Yaskawa INFORM job: X2_29-32(-90,180)_HARDOX.JBI

/JOB
//NAME X2_29-32(-90,180)_HARDOX
//POS
///NPOS 464,464,464,30,0,0
///TOOL 0
///POSTYPE PULSE
///PULSE
C00000=2000,-95440,-72516,0,38121,0
C00001=-80443,-95440,-72516,-46202,38121,50067
C00002=-52411,-63190,-65629,-41206,65263,51508
C00003=-73087,-23788,-54178,-20049,70640,39353
C00004=-137855,-58890,-63164,50426,57117,3007
C00005=-121629,-1819,-23267,32035,72941,16834
C00006=-120935,3126,-16373,32060,71231,16611
C00007=-120668,5150,-13541,32087,70531,16512
C00008=-120826,7275,-11699,32150,70554,16454
C00009=-120668,5150,-13541,32087,70531,16512
C00010=-120649,6560,-12069,32112,70369,16472
C00011=-120645,6560,-10825,32251,69714,16277
C00012=-120649,6560,-12069,32112,70369,16472
C00013=-120913,4529,-14922,32082,71075,16573
C00014=-121602,-429,-21862,32048,72802,16805
C00015=-120074,-1541,-23154,10906,71264,22392
C00016=-120462,3262,-16191,11181,69532,22093
C00017=-120612,5232,-13331,11295,68818,21971
C00018=-120770,7357,-11488,11363,68799,21912
C00019=-120612,5232,-13331,11295,68818,21971
C00020=-120702,6360,-12382,11332,68826,21940
C00021=-120699,6356,-11141,11388,68075,21868
C00022=-120702,6360,-12382,11332,68826,21940
C00023=-120555,4389,-15254,11219,69547,22062
C00024=-120172,-412,-22245,10944,71297,22361
C00025=-149351,-10161,-47708,21219,87013,14604
C00026=-137351,69022,23166,10145,93880,-87530
C00027=-140356,69806,28572,10729,91371,-88714
C00028=-140356,69507,29335,10724,90759,-88767
C00029=-140356,69553,29212,10724,90856,-88758
C00030=-140261,66601,25742,10710,91452,-88676
C00031=-140356,69553,29212,10724,90856,-88758
C00032=-136478,56234,14982,2602,86089,-89060
C00033=-137167,55940,14650,2804,86164,-89279
C00034=-140356,69877,28402,10731,91510,-88702
C00035=-138692,40861,2416,14344,76332,-89060
C00036=-138692,40492,3371,14387,75578,-89150
C00037=-138692,40531,3265,14382,75660,-89140
C00038=-138845,42877,5737,14463,75381,-89226
C00039=-138692,40531,3265,14382,75660,-89140
C00040=-137711,40836,3584,13981,75458,-88832
C00041=-137936,41046,2771,14040,76086,-88835
C00042=-125437,22929,-16002,8654,76643,-84658
C00043=-125437,22691,-15519,8668,76228,-84687
C00044=-125436,22336,-14745,8692,75581,-84731
C00045=-125436,22385,-14855,8689,75673,-84725
C00046=-125647,22419,-14823,8780,75693,-84793
C00047=-125456,22816,-15761,8671,76446,-84677
C00048=-124626,66836,21249,8312,76213,-84427
C00049=-124626,66325,22111,8339,75427,-84480
C00050=-124626,66371,22030,8336,75501,-84476
C00051=-124784,66398,22063,8405,75510,-84527
C00052=-124718,66903,21186,8350,76294,-84452
C00053=-140356,71956,24660,10787,94825,-88416
C00054=-145256,112136,75534,11701,85011,-90920
C00055=-134601,86997,59569,9608,80583,-87665
C00056=-133445,96084,71731,8965,80046,-87331
C00057=-133445,96731,74588,9003,78636,-87434
C00058=-133445,96669,74335,9000,78758,-87425
C00059=-133228,92094,68499,8930,79959,-87263
C00060=-133445,96669,74335,9000,78758,-87425
C00061=-133796,95310,72593,9053,79166,-87516
C00062=-134289,94368,71392,9135,79474,-87664
C00063=-133445,96257,72553,8977,79632,-87361
C00064=-124701,59773,45425,12728,59446,-85623
C00065=-124701,60369,47958,12892,58224,-85768
C00066=-124701,60307,47711,12875,58342,-85755
C00067=-125124,62964,50756,13140,57912,-85979
C00068=-124701,60307,47711,12875,58342,-85755
C00069=-124156,61205,48739,12645,58092,-85564
C00070=-123633,62204,49884,12428,57822,-85386
C00071=-124701,59815,45622,12740,59350,-85635
C00072=-140824,71424,26731,-14708,78728,-67313
C00073=-138566,88921,46332,-15736,76162,-66229
C00074=-147570,88381,37329,-2994,91316,-68707
C00075=-150504,94687,46185,-534,91721,-69351
C00076=-150504,94129,46947,-534,90966,-69348
C00077=-150505,94206,46833,-534,91077,-69347
C00078=-150278,92960,45244,-584,91415,-69274
C00079=-150242,94003,44864,-592,92185,-69267
C00080=-154498,83968,32184,366,94826,-70609
C00081=-154498,83134,33047,365,93865,-70611
C00082=-154498,83201,32975,365,93945,-70611
C00083=-154422,82409,31994,348,94142,-70584
C00084=-154454,83590,32320,355,94549,-70593
C00085=-163409,96576,47553,1962,92625,-73499
C00086=-157730,108398,64416,-12689,90385,-74066
C00087=-157730,108035,65300,-12685,89672,-73993
C00088=-157730,108081,65179,-12685,89767,-74003
C00089=-157935,107012,63772,-12649,90048,-74099
C00090=-157741,107169,62938,-12691,90658,-74096
C00091=-153583,44731,-17162,-14334,108038,-74686
C00092=-119941,-49108,-60020,12756,52739,20459
C00093=-119789,-74783,-79746,11606,60570,21449
C00094=-121427,-115493,-86071,-971,23186,13
C00095=-103613,-33005,-61039,-35202,65094,-22685
C00096=-106311,42726,-13762,-25892,102641,-65108
C00097=-107595,62330,8123,-25246,99218,-64778
C00098=-113201,64656,7277,-4573,99753,-62165
C00099=-113587,63448,8349,-4464,98459,-62235
C00100=-113587,62765,8896,-4459,97772,-62209
C00101=-113587,62841,8834,-4460,97849,-62212
C00102=-113249,60648,6293,-4545,98301,-62127
C00103=-113587,62841,8834,-4460,97849,-62212
C00104=-104619,65495,14505,-22863,97888,-62863
C00105=-105135,64543,13388,-22764,97939,-63047
C00106=-113587,63726,8142,-4473,98728,-62244
C00107=-108677,35532,-14553,-8240,80429,-60363
C00108=-108677,34745,-13725,-8259,79524,-60302
C00109=-108677,34861,-13853,-8256,79661,-60312
C00110=-109185,36959,-11698,-8032,79365,-60451
C00111=-108678,34861,-13851,-8256,79664,-60311
C00112=-108199,35754,-12936,-8475,79600,-60161
C00113=-107535,36718,-11943,-8775,79549,-59951
C00114=-108678,35482,-14504,-8241,80378,-60358
C00115=-107675,14693,-34978,-8652,82358,-60193
C00116=-103613,-33005,-61039,-35202,65094,-22685
C00117=-118652,-1130,-18887,-50959,75871,-22344
C00118=-120065,3095,-12579,-50928,73991,-22034
C00119=-120612,5858,-10323,-50783,73711,-22168
C00120=-120794,7716,-8707,-50742,73586,-22192
C00121=-120612,6719,-9575,-50786,73699,-22162
C00122=-120612,6754,-8612,-50907,73330,-21953
C00123=-120612,6719,-9575,-50786,73699,-22162
C00124=-120164,4326,-11494,-50910,73914,-22043
C00125=-118762,92,-17836,-50934,75798,-22362
C00126=-120082,-2017,-23568,-21020,76850,-12939
C00127=-120471,2786,-16617,-21041,75059,-12760
C00128=-120621,6055,-13261,-21027,74660,-12744
C00129=-120866,7545,-11965,-20950,74569,-12818
C00130=-120698,6523,-12855,-21003,74632,-12768
C00131=-120698,6506,-12245,-21039,74273,-12705
C00132=-120698,6523,-12855,-21003,74632,-12768
C00133=-120547,3972,-15593,-21018,75020,-12781
C00134=-120163,-831,-22574,-20994,76828,-12964
C00135=-120068,-2141,-23641,-4094,79360,4817
C00136=-120458,2664,-16692,-4000,77538,4745
C00137=-120609,5664,-13523,-3960,77123,4708
C00138=-120915,7025,-12341,-3868,77081,4605
C00139=-120609,5664,-13523,-3960,77123,4708
C00140=-120609,5646,-12752,-3962,76640,4725
C00141=-120609,5664,-13523,-3960,77123,4708
C00142=-120559,4206,-15421,-3970,77544,4711
C00143=-120175,-595,-22406,-4061,79389,4780
C00144=-120687,14813,-21149,-8531,87328,5298
C00145=-120686,13947,-18988,-8540,85572,5418
C00146=-121162,15330,-17687,-8405,85435,5272
C00147=-120827,14308,-18485,-8500,85444,5381
C00148=-120926,18777,-11948,-23218,84672,-11491
C00149=-120686,12805,-15419,-25390,80631,-12632
C00150=-120686,13423,-17789,-25296,82244,-12980
C00151=-103613,-33005,-61039,-35202,65094,-22685
C00152=-106311,42726,-13762,-25892,102641,-65108
C00153=-107595,62330,8123,-25246,99218,-64778
C00154=-113201,64656,7277,-4573,99753,-62165
C00155=-140379,75416,22801,13293,101526,-67991
C00156=-140410,74339,22937,13264,100908,-68069
C00157=-136164,75986,24927,12542,99919,-66800
C00158=-136164,75986,24927,12542,99919,-66800
C00159=-130307,51965,-280,1869,88480,-68213
C00160=-130096,37123,-11525,-190,78489,-68727
C00161=-129173,33980,-14136,-6116,77606,-69795
C00162=-117721,30667,-17043,-13656,78654,-66867
C00163=-117721,30667,-17043,-13656,78654,-66867
C00164=-116349,51111,-1470,-15144,92480,-68252
C00165=-140410,74339,22937,13264,100908,-68069
C00166=-140394,75226,22544,13300,101585,-67989
C00167=-143024,47479,-9541,14128,107315,-68172
C00168=-103613,-33005,-61039,-35202,65094,-22685
C00169=-121427,-115493,-86071,-971,23186,13
C00170=-119789,-74783,-79746,11606,60570,21449
C00171=-119941,-49108,-60020,12756,52739,20459
C00172=-140276,36725,370,11673,88260,-76470
C00173=-134601,86997,59569,9608,80583,-87665
C00174=-138207,103684,77785,17301,84049,-88284
C00175=-137334,101091,76947,17225,83081,-88111
C00176=-133753,108880,87117,16824,80164,-87228
C00177=-133753,108880,87117,16824,80164,-87228
C00178=-134207,73969,56380,20261,66539,-89438
C00179=-133045,60996,43275,16271,60703,-90304
C00180=-131571,55694,36295,8271,61065,-90068
C00181=-118397,49989,30000,-2055,61299,-85309
C00182=-118397,49989,30000,-2055,61299,-85309
C00183=-130531,95421,68229,8568,83299,-86105
C00184=-137334,101091,76947,17225,83081,-88111
C00185=-137309,103311,78077,17211,83503,-88042
C00186=-146018,96073,47329,18619,99857,-88679
C00187=-146906,94555,49940,18578,97784,-89305
C00188=-142933,95333,50973,18069,96712,-88106
C00189=-142933,95333,50973,18069,96712,-88106
C00190=-142636,61819,14681,18419,84430,-90138
C00191=-141138,57519,10350,14135,81366,-90943
C00192=-124192,48626,472,-4337,80868,-88195
C00193=-120975,45190,-1140,-14592,79533,-89080
C00194=-120975,45190,-1140,-14592,79533,-89080
C00195=-121205,42490,-4021,-14479,79869,-89194
C00196=-146906,94555,49940,18578,97784,-89305
C00197=-146868,95992,48950,18656,99055,-89096
C00198=-148689,99526,52175,12058,97492,78019
C00199=-152884,101141,55717,10807,87410,75244
C00200=-156822,87647,42567,16335,79952,73793
C00201=-156347,101107,61134,16633,80023,73987
C00202=-156384,100515,60368,16637,80191,73997
C00203=-156384,100515,60368,16637,80191,73997
C00204=-156439,104263,64294,16482,82615,74284
C00205=-153753,110748,70719,9837,85116,74669
C00206=-150674,104620,59635,-3355,94991,76839
C00207=-155137,96651,49130,-4365,100310,75004
C00208=-155137,96651,49130,-4365,100310,75004
C00209=-157583,94336,46084,-1766,101365,64930
C00210=-158276,84861,34738,-3244,98222,56321
C00211=-159116,67672,17693,-4464,87885,55617
C00212=-158508,68290,14812,-4659,90001,55728
C00213=-159737,63424,5379,-4280,93236,55245
C00214=-162760,44138,-13287,27476,96226,62089
C00215=-135421,18423,-39272,17962,92414,69811
C00216=-134350,548,-53000,17534,91515,69996
C00217=-134346,591,-47047,17501,88033,69498
C00218=-133581,11899,-36465,17450,85821,69480
C00219=-133633,12580,-37298,17464,86638,69580
C00220=-133478,14153,-35291,17454,85907,69536
C00221=-130266,45661,-10200,12167,104064,71599
C00222=-133264,15600,-32829,17378,85127,69491
C00223=-130716,70167,29007,18289,68146,68029
C00224=-130765,70515,28279,18240,68753,68107
C00225=-130672,73101,31358,18260,68194,68051
C00226=-130688,71478,30626,18340,67728,67974
C00227=-130258,88127,52093,19258,61489,67116
C00228=-130258,88603,49705,18973,63112,67401
C00229=-136006,-18137,-67664,18160,91268,69467
C00230=-130548,-59686,-65936,20231,53139,15983
C00231=-120686,14413,-19191,15888,76861,21657
C00232=-120686,13677,-16924,15998,75153,21431
C00233=-120864,13854,-15557,16118,74464,21280
C00234=-120686,13319,-15964,16052,74414,21331
C00235=-120685,12972,2532,58159,63782,21773
C00236=-120685,12849,1627,57961,64053,21984
C00237=-120685,12557,-1021,57383,64873,22611
C00238=-118042,2496,-28680,21493,77866,23942
C00239=-119941,-49108,-60020,12756,52739,20459
C00240=-119789,-74783,-79746,11606,60570,21449
C00241=-121427,-115493,-86071,-971,23186,13
C00242=-103613,-33005,-61039,-35202,65094,-22685
C00243=-134099,37898,13128,-30528,62935,-29291
C00244=-134100,37844,14655,-30775,62096,-29040
C00245=-131820,39720,18358,-33617,61933,-27865
C00246=-133865,38946,16955,-31235,61462,-28734
C00247=-133724,38989,23896,-55752,81870,-5528
C00248=-134106,38309,22847,-57056,83615,-3951
C00249=-130543,37429,19989,-57378,86491,-3781
C00250=-124532,-28339,-37080,2656,37858,63256
C00251=-80443,-95440,-72516,-46202,38121,50067
C00252=-628,-74499,-67639,-57475,89722,72456
C00253=3643,-76224,-106676,19950,71810,76872
C00254=-57022,-39792,-97587,-14580,73098,62715
C00255=-77894,6609,-39652,-10081,68656,55583
C00256=-79326,8848,-34628,-9340,66588,55287
C00257=-79882,9812,-32559,-9051,65763,55166
C00258=-80655,11957,-30643,-8578,65611,54918
C00259=-79882,9812,-32559,-9051,65763,55166
C00260=-80541,11612,-30977,-8647,65649,54954
C00261=-80539,10894,-29907,-8717,64633,55031
C00262=-80541,11612,-30977,-8647,65649,54954
C00263=-79996,10638,-33064,-8931,66478,55073
C00264=-78593,8374,-38132,-9661,68553,55366
C00265=-77879,6415,-39661,-10096,68566,55596
C00266=-79312,8664,-34633,-9354,66499,55298
C00267=-79868,9631,-32562,-9065,65674,55178
C00268=-80642,11778,-30647,-8592,65523,54929
C00269=-79868,9631,-32562,-9065,65674,55178
C00270=-80486,11377,-31039,-8686,65573,54978
C00271=-80483,10662,-29965,-8757,64557,55056
C00272=-80486,11377,-31039,-8686,65573,54978
C00273=-79940,10400,-33127,-8971,66401,55097
C00274=-78534,8129,-38197,-9702,68474,55392
C00275=-80101,2636,-42462,-8765,68121,54914
C00276=-81514,5018,-37368,-8012,66098,54596
C00277=-82062,6036,-35274,-7718,65291,54467
C00278=-82824,8247,-33345,-7247,65177,54218
C00279=-82062,6036,-35274,-7718,65291,54467
C00280=-82687,7884,-33751,-7328,65251,54260
C00281=-82684,7173,-32662,-7390,64223,54326
C00282=-82687,7884,-33751,-7328,65251,54260
C00283=-82150,6860,-35861,-7618,66062,54387
C00284=-80765,4464,-40992,-8359,68092,54701
C00285=-102565,-17528,-58279,5105,67037,47705
C00286=-103540,-14129,-52689,5779,65410,47308
C00287=-103914,-12731,-50412,6044,64755,47149
C00288=-104433,-9984,-48291,6364,64897,46981
C00289=-103914,-12731,-50412,6044,64755,47149
C00290=-104359,-10402,-48741,6314,64954,47009
C00291=-104354,-11138,-47602,6366,63880,46952
C00292=-104359,-10402,-48741,6314,64954,47009
C00293=-103995,-11787,-51026,6054,65619,47167
C00294=-103047,-15149,-56634,5395,67274,47560
C00295=-80233,11979,-33534,-13378,69985,55632
C00296=-80229,10556,-31784,-13533,68226,55836
C00297=-80227,10062,-31089,-13596,67561,55913
C00298=-85904,3072,-37201,-10254,66968,54061
C00299=-91604,-2565,-41777,-6847,66341,52198
C00300=-101176,-9655,-47350,-1032,65699,49019
C00301=-100886,-9155,-48096,-1203,66417,49108
C00302=-100216,-7271,-49632,-1590,68341,49304
C00303=-80300,11336,-32181,-3939,63811,54132
C00304=-80297,10024,-30348,-4003,62013,54196
C00305=-80296,9579,-29637,-4028,61349,54220
C00306=-80356,9883,-29495,-3999,61418,54197
C00307=-80338,10281,-30338,-3972,62137,54177
C00308=-80341,11605,-32161,-3909,63935,54114
C00309=-57022,-39792,-97587,-14580,73098,62715
C00310=-628,-74499,-67639,-57475,89722,72456
C00311=-628,-74499,-67639,-57475,89722,72456
C00312=-616,-75233,-71189,-57531,90735,71761
C00313=3643,-76224,-106674,19950,71813,76873
C00314=-42730,11015,-70691,-38334,96086,2936
C00315=-63606,9545,-60534,-45336,92087,-16638
C00316=-78956,5069,-41799,-36523,82652,-30708
C00317=-79715,8164,-36018,-36343,80767,-30358
C00318=-80007,9457,-33651,-36288,80012,-30216
C00319=-80417,12097,-31285,-36126,79775,-30292
C00320=-80007,9457,-33651,-36288,80012,-30216
C00321=-80344,11698,-31669,-36153,79828,-30282
C00322=-80337,10939,-30633,-36254,78993,-30001
C00323=-80344,11698,-31669,-36153,79828,-30282
C00324=-80059,10405,-34052,-36203,80590,-30428
C00325=-79319,7312,-39869,-36371,82488,-30786
C00326=-78994,5332,-41692,-36502,82694,-30736
C00327=-79751,8420,-35912,-36322,80808,-30385
C00328=-80043,9710,-33546,-36267,80051,-30242
C00329=-80452,12349,-31177,-36105,79813,-30317
C00330=-80043,9710,-33546,-36267,80051,-30242
C00331=-80378,11838,-31671,-36133,79874,-30310
C00332=-80371,11075,-30637,-36233,79039,-30029
C00333=-80378,11838,-31671,-36133,79874,-30310
C00334=-80093,10547,-34052,-36183,80637,-30456
C00335=-79355,7462,-39866,-36352,82536,-30815
C00336=-79090,5824,-41546,-36452,82791,-30803
C00337=-79842,8894,-35770,-36272,80900,-30451
C00338=-80133,10177,-33405,-36216,80142,-30307
C00339=-80539,12815,-31031,-36055,79902,-30380
C00340=-80133,10177,-33405,-36216,80142,-30307
C00341=-80467,12378,-31515,-36079,79989,-30382
C00342=-80461,11606,-30490,-36178,79153,-30101
C00343=-80467,12378,-31515,-36079,79989,-30382
C00344=-80184,11095,-33894,-36130,80753,-30529
C00345=-79450,8031,-39703,-36300,82657,-30890
C00346=-79130,5997,-41490,-36432,82820,-30827
C00347=-79881,9061,-35715,-36251,80928,-30474
C00348=-80171,10342,-33350,-36196,80169,-30330
C00349=-80577,12980,-30974,-36035,79928,-30403
C00350=-80171,10342,-33350,-36196,80169,-30330
C00351=-80499,12601,-31443,-36059,80034,-30409
C00352=-80493,11826,-30422,-36158,79199,-30129
C00353=-80499,12601,-31443,-36059,80034,-30409
C00354=-80216,11321,-33822,-36110,80799,-30556
C00355=-79484,8265,-39628,-36281,82705,-30918
C00356=-80360,13355,-34008,-31162,79863,-31191
C00357=-80358,11846,-32319,-31320,78301,-30757
C00358=-80129,11573,-31352,-31494,77744,-30518
C00359=-80458,11751,-31298,-31342,77685,-30622
C00360=-80398,12063,-32232,-31297,78337,-30782
C00361=-80400,13577,-33916,-31139,79899,-31215
C00362=-80289,11819,-32883,-40833,82428,-30239
C00363=-80286,10439,-31086,-40975,81039,-29694
C00364=-80284,9940,-30341,-41041,80492,-29477
C00365=-80262,9799,-30343,-41055,80447,-29451
C00366=-80245,10226,-31168,-40996,81011,-29666
C00367=-80248,11601,-32971,-40853,82401,-30212
C00368=-66712,19655,-58640,-43457,90055,-24381
C00369=-33423,17994,-60377,-60627,102988,-19600
C00370=-628,-74499,-67639,-57475,89722,-77289
C00371=-111516,-94989,-87682,-11539,41033,-8318
C00372=-107125,-12532,-46236,-32676,64375,-10703
C00373=-119952,37605,6162,-31233,75137,-17424
C00374=-120511,42562,14108,-31354,72919,-17016
C00375=-120728,44654,17433,-31427,72005,-16841
C00376=-120598,46946,19889,-31526,71766,-16719
C00377=-120728,44654,17433,-31427,72005,-16841
C00378=-120690,45788,18679,-31469,71861,-16784
C00379=-120687,45721,19851,-31594,71213,-16595
C00380=-120690,45788,18679,-31469,71861,-16784
C00381=-120474,43679,15324,-31394,72783,-16962
C00382=-119917,38688,7316,-31265,75018,-17376
C00383=-121235,29127,929,-10497,72605,-22385
C00384=-120892,33963,8709,-10768,70384,-22067
C00385=-120760,35995,11952,-10883,69467,-21936
C00386=-120625,38237,14258,-10956,69222,-21864
C00387=-120760,35995,11952,-10883,69467,-21936
C00388=-120657,37146,13206,-10937,69303,-21884
C00389=-120654,37124,14427,-10991,68554,-21813
C00390=-120657,37146,13206,-10937,69303,-21884
C00391=-120788,35099,9935,-10821,70230,-22016
C00392=-121127,30229,2096,-10548,72470,-22335
C00393=-114017,-48711,-62992,-16459,47417,-13874
C00394=-111516,-94989,-87682,-11539,41033,-8318
C00395=-126605,-77887,-93073,32833,63422,15189
C00396=-122507,12852,-43627,17515,100315,22769
C00397=-122731,-562,-19309,51196,76332,22742
C00398=-121309,3590,-13049,51151,74446,22427
C00399=-120759,5312,-10468,51156,73690,22291
C00400=-120602,7442,-8613,51127,73573,22309
C00401=-120759,5312,-10468,51156,73690,22291
C00402=-120666,6547,-9361,51143,73609,22295
C00403=-120662,6597,-8073,51308,73115,22013
C00404=-120666,6547,-9361,51143,73609,22295
C00405=-121212,4820,-11958,51134,74367,22434
C00406=-122622,659,-18251,51172,76257,22758
C00407=-122507,10859,-42333,17402,98575,22516
C00408=-121302,-1391,-23074,21379,77148,13095
C00409=-120901,3377,-16122,21398,75339,12912
C00410=-120747,5333,-13267,21416,74597,12833
C00411=-120590,7459,-11416,21370,74514,12875
C00412=-120747,5333,-13267,21416,74597,12833
C00413=-120673,6521,-12221,21396,74547,12851
C00414=-120670,6504,-10992,21468,73832,12721
C00415=-120673,6521,-12221,21396,74547,12851
C00416=-120826,4563,-15090,21376,75296,12931
C00417=-121222,-206,-22073,21354,77121,13119
C00418=-121314,-1652,-23262,4485,79740,-4708
C00419=-120913,3117,-16316,4391,77900,-4639
C00420=-120758,5074,-13462,4356,77144,-4613
C00421=-120601,7199,-11615,4311,77090,-4561
C00422=-120758,5074,-13462,4356,77144,-4613
C00423=-120661,6618,-12165,4328,77134,-4580
C00424=-120658,6600,-10936,4339,76370,-4606
C00425=-120661,6618,-12165,4328,77134,-4580
C00426=-120814,4660,-15035,4362,77900,-4605
C00427=-121209,-107,-22019,4454,79763,-4672
C00428=-120687,46979,12625,8958,83453,-5452
C00429=-120687,46939,12852,8960,83294,-5464
C00430=-121610,47377,14332,9229,82719,-5809
C00431=-120687,46779,13614,8967,82756,-5503
C00432=-120687,46744,18453,25999,77793,12121
C00433=-120687,46348,16793,25935,78533,12285
C00434=-120687,46750,14296,25811,80109,12635
C00435=-133650,-5326,-40947,35821,67459,4738
C00436=-126605,-79487,-84548,34660,58331,13454
C00437=-111516,-94989,-87682,-11539,41033,-8318
C00438=-114017,-48711,-62992,-16459,47417,-13874
C00439=-117875,8541,-26754,-15356,68464,-18868
C00440=-120687,46680,12303,-15684,74586,-21239
C00441=-120687,46183,14573,-15804,72993,-21028
C00442=-120687,45847,15503,-15862,72274,-20933
C00443=-120687,45820,15711,-15860,72146,-20914
C00444=-120686,46430,31549,-51889,62431,-21622
C00445=-120686,46225,30262,-51616,62867,-21897
C00446=-120686,45862,27317,-50999,63909,-22538
C00447=-117875,8541,-26754,-15356,68464,-18868
C00448=-114017,-48711,-62992,-16459,47417,-13874
C00449=-111516,-94989,-87682,-11539,41033,-8318
C00450=-126605,-79487,-84548,34660,58331,13454
C00451=-133650,-5326,-40947,35821,67459,4738
C00452=-107292,16964,-8341,30286,65218,30077
C00453=-107291,16711,-5651,30703,63668,29626
C00454=-107319,17056,-4163,30899,63039,29427
C00455=-107325,17150,-4064,30903,63037,29424
C00456=-107531,17120,3962,56911,83437,5110
C00457=-107292,16975,3345,57479,84239,4502
C00458=-107292,16775,1094,57407,84952,4997
C00459=-118083,23631,-28824,25815,115568,5891
C00460=-116334,-45445,-82386,24519,90130,1359
C00461=-114916,-111439,-107393,23774,54945,-5331
C00462=-628,-74499,-67639,-57475,89722,-77289
C00463=2000,17994,-60377,0,102988,0
BC00000=30861,666204,744559
BC00001=125925,693938,117612
BC00002=171995,715848,96803
BC00003=199966,729151,84169
BC00004=289373,771673,43785
BC00005=289373,771673,43785
BC00006=289373,771673,43785
BC00007=289373,771673,43785
BC00008=289373,771673,43785
BC00009=289373,771673,43785
BC00010=289373,771673,43785
BC00011=289373,771673,43785
BC00012=289373,771673,43785
BC00013=289373,771673,43785
BC00014=289373,771673,43785
BC00015=275430,758658,78312
BC00016=275430,758658,78312
BC00017=275430,758658,78312
BC00018=275430,758658,78312
BC00019=275430,758658,78312
BC00020=275430,758658,78312
BC00021=275430,758658,78312
BC00022=275430,758658,78312
BC00023=275430,758658,78312
BC00024=275430,758658,78312
BC00025=343308,785974,78310
BC00026=343308,785974,78310
BC00027=343308,785974,78310
BC00028=343308,785974,78310
BC00029=343308,785974,78310
BC00030=343308,785974,78310
BC00031=343308,785974,78310
BC00032=343308,785974,78310
BC00033=343308,785974,78310
BC00034=343308,785974,78310
BC00035=343308,785974,78310
BC00036=343308,785974,78310
BC00037=343308,785974,78310
BC00038=343308,785974,78310
BC00039=343308,785974,78310
BC00040=343308,785974,78310
BC00041=343308,785974,78310
BC00042=318074,785974,78310
BC00043=318074,785974,78310
BC00044=318074,785974,78309
BC00045=318074,785974,78309
BC00046=318074,785974,78309
BC00047=318074,785974,78309
BC00048=318074,785624,15543
BC00049=318074,785624,15543
BC00050=318074,785624,15543
BC00051=318074,785624,15543
BC00052=318074,785624,15543
BC00053=343308,785974,78310
BC00054=370182,760337,78310
BC00055=370182,760337,184963
BC00056=370182,760337,157808
BC00057=370182,760337,157808
BC00058=370182,760337,157808
BC00059=370182,760337,157808
BC00060=370182,760337,157808
BC00061=370182,760337,157808
BC00062=370182,760337,157808
BC00063=370182,760337,157808
BC00064=340749,760337,227440
BC00065=340749,760337,227440
BC00066=340749,760337,227440
BC00067=340749,760337,227440
BC00068=340749,760337,227440
BC00069=340749,760337,227440
BC00070=340749,760337,227440
BC00071=340749,760337,227440
BC00072=340750,760338,77389
BC00073=340750,760338,30516
BC00074=348215,785472,13
BC00075=348215,785472,13
BC00076=348215,785471,10
BC00077=348215,785471,9
BC00078=348215,785471,9
BC00079=348215,785471,9
BC00080=348215,785471,9
BC00081=348215,785471,9
BC00082=348215,785471,9
BC00083=348215,785471,9
BC00084=348215,785471,9
BC00085=370537,785471,9
BC00086=370537,785471,9
BC00087=370537,785471,9
BC00088=370537,785471,9
BC00089=370537,785471,9
BC00090=370537,785471,9
BC00091=370537,785471,9
BC00092=275430,725446,78312
BC00093=275430,674753,78312
BC00094=160005,679271,117612
BC00095=134493,734471,53
BC00096=134493,734471,4
BC00097=134493,734471,4
BC00098=134493,734471,4
BC00099=134493,734471,4
BC00100=134493,734471,4
BC00101=134493,734471,4
BC00102=134493,734471,4
BC00103=134493,734471,4
BC00104=134493,734471,4
BC00105=134493,734471,4
BC00106=134493,734471,4
BC00107=134493,734471,4
BC00108=134493,734471,4
BC00109=134493,734471,4
BC00110=134493,734471,4
BC00111=134494,734471,1
BC00112=134493,734471,4
BC00113=134493,734471,4
BC00114=134494,734471,1
BC00115=134493,734471,4
BC00116=134493,734471,53
BC00117=134493,734471,53
BC00118=134493,734471,53
BC00119=134493,734471,53
BC00120=134493,734471,53
BC00121=134493,734471,53
BC00122=134493,734471,53
BC00123=134493,734471,53
BC00124=134493,734471,53
BC00125=134493,734471,53
BC00126=120013,731989,63282
BC00127=120013,731989,63282
BC00128=120013,731989,63282
BC00129=120013,731989,63282
BC00130=120013,731989,63282
BC00131=120013,731989,63282
BC00132=120013,731989,63282
BC00133=120013,731989,63282
BC00134=120013,731989,63282
BC00135=143296,743099,87341
BC00136=143296,743099,87341
BC00137=143296,743099,87341
BC00138=143296,743099,87341
BC00139=143296,743099,87341
BC00140=143296,743099,87341
BC00141=143296,743099,87341
BC00142=143296,743099,87341
BC00143=143296,743099,87341
BC00144=160875,733218,0
BC00145=159215,738452,0
BC00146=159050,738970,0
BC00147=154263,739676,0
BC00148=124438,729775,0
BC00149=121804,726587,0
BC00150=123464,721353,0
BC00151=134493,734471,53
BC00152=134493,734471,4
BC00153=134493,734471,4
BC00154=134493,734471,4
BC00155=202496,734468,2
BC00156=202496,734468,2
BC00157=202496,734468,2
BC00158=202496,734468,2
BC00159=202496,734468,2
BC00160=202496,734468,2
BC00161=202496,734468,2
BC00162=167019,734468,2
BC00163=167019,734468,2
BC00164=163805,734468,2
BC00165=202496,734468,2
BC00166=202496,734468,2
BC00167=202496,734468,2
BC00168=134493,734471,53
BC00169=160005,679271,117612
BC00170=275430,674753,78312
BC00171=275430,725446,78312
BC00172=359023,756228,172403
BC00173=370182,760337,184963
BC00174=370182,760337,129528
BC00175=370181,760337,129525
BC00176=370055,760318,129428
BC00177=370055,760318,129428
BC00178=370055,760499,186673
BC00179=370055,760499,186673
BC00180=369975,760487,186584
BC00181=327884,760487,186584
BC00182=327884,760487,186584
BC00183=355542,760337,129525
BC00184=370181,760337,129525
BC00185=370181,760337,129525
BC00186=355947,779528,6445
BC00187=356286,779072,9376
BC00188=356321,779025,9678
BC00189=356321,779025,9678
BC00190=356321,779025,9678
BC00191=356321,779025,9727
BC00192=316277,778464,10141
BC00193=316277,778464,10141
BC00194=316277,778464,10141
BC00195=316277,778464,10141
BC00196=356286,779072,9376
BC00197=356286,779072,9376
BC00198=356286,779072,9376
BC00199=356286,779072,9376
BC00200=356286,779072,9376
BC00201=356286,779072,9376
BC00202=356286,779072,9376
BC00203=356286,779072,9376
BC00204=356286,779072,9376
BC00205=356286,779072,9376
BC00206=359300,795873,31
BC00207=359300,795873,31
BC00208=359300,795873,31
BC00209=359300,795873,31
BC00210=359300,795873,31
BC00211=359300,795873,31
BC00212=359300,795873,31
BC00213=359300,795873,31
BC00214=359300,795873,31
BC00215=329302,795872,29
BC00216=329302,795872,29
BC00217=329302,795872,29
BC00218=329622,793366,28
BC00219=329626,793338,28
BC00220=329692,792815,28
BC00221=329692,792815,28
BC00222=329692,792815,28
BC00223=331278,780389,22
BC00224=331278,780389,22
BC00225=331278,780389,22
BC00226=331302,780203,22
BC00227=331702,777069,20
BC00228=331702,777069,20
BC00229=329302,795872,29
BC00230=311672,797875,78800
BC00231=261630,745054,0
BC00232=261335,750526,0
BC00233=262635,752963,0
BC00234=310200,761264,0
BC00235=269037,768534,0
BC00236=267560,766459,0
BC00237=263869,761272,0
BC00238=263869,761272,0
BC00239=275430,725446,78312
BC00240=275430,674753,78312
BC00241=160005,679271,117612
BC00242=134493,734471,53
BC00243=177141,688062,0
BC00244=175480,693296,0
BC00245=174817,695179,178
BC00246=160472,692881,15
BC00247=152915,732429,1
BC00248=154775,734615,0
BC00249=161011,731782,0
BC00250=160005,693938,117612
BC00251=125925,693938,117612
BC00252=97174,666880,426359
BC00253=199464,674570,1075173
BC00254=48447,721710,1061717
BC00255=196183,770700,1075175
BC00256=196183,770700,1075175
BC00257=196183,770700,1075175
BC00258=196183,770700,1075175
BC00259=196183,770700,1075175
BC00260=196183,770700,1075175
BC00261=196183,770700,1075175
BC00262=196183,770700,1075175
BC00263=196183,770700,1075175
BC00264=196183,770700,1075175
BC00265=139869,760824,1075175
BC00266=139869,760824,1075175
BC00267=139869,760824,1075175
BC00268=139869,760824,1075175
BC00269=139869,760824,1075175
BC00270=139869,760824,1075175
BC00271=139869,760824,1075175
BC00272=139869,760824,1075175
BC00273=139869,760824,1075175
BC00274=139869,760824,1075175
BC00275=15,735270,1075175
BC00276=15,735270,1075175
BC00277=15,735270,1075175
BC00278=15,735270,1075175
BC00279=15,735270,1075175
BC00280=15,735270,1075175
BC00281=15,735270,1075175
BC00282=15,735270,1075175
BC00283=15,735270,1075175
BC00284=15,735270,1075175
BC00285=15,725270,1075175
BC00286=15,725270,1075175
BC00287=15,725270,1075175
BC00288=15,725270,1075175
BC00289=15,725270,1075175
BC00290=15,725270,1075175
BC00291=15,725270,1075175
BC00292=15,725270,1075175
BC00293=15,725270,1075175
BC00294=15,725270,1075175
BC00295=12536,730414,1075175
BC00296=10876,735648,1075175
BC00297=10211,737741,1075175
BC00298=7204,734292,1075175
BC00299=4400,731075,1075175
BC00300=15,726043,1075175
BC00301=15,723950,1075175
BC00302=15,718716,1075175
BC00303=125627,754347,1075175
BC00304=125333,759820,1075175
BC00305=125215,762009,1075175
BC00306=192338,773707,1075173
BC00307=192456,771518,1075175
BC00308=192751,766045,1075175
BC00309=48447,721710,1061717
BC00310=97174,666880,1005640
BC00311=97174,666880,842388
BC00312=97174,666880,900747
BC00313=199464,674570,1075172
BC00314=79996,736581,994878
BC00315=45352,753605,1043201
BC00316=33984,772629,1075175
BC00317=33984,772629,1075175
BC00318=33984,772629,1075175
BC00319=33984,772629,1075175
BC00320=33984,772629,1075175
BC00321=33984,772629,1075175
BC00322=33984,772629,1075175
BC00323=33984,772629,1075175
BC00324=33984,772629,1075175
BC00325=33984,772629,1075175
BC00326=90316,762849,1075175
BC00327=90316,762849,1075175
BC00328=90316,762849,1075175
BC00329=90316,762849,1075175
BC00330=90316,762849,1075175
BC00331=90316,762849,1075175
BC00332=90316,762849,1075175
BC00333=90316,762849,1075175
BC00334=90316,762849,1075175
BC00335=90316,762849,1075175
BC00336=237131,737545,1075175
BC00337=237131,737545,1075175
BC00338=237131,737545,1075175
BC00339=237131,737545,1075175
BC00340=237131,737545,1075175
BC00341=237131,737545,1075175
BC00342=237131,737545,1075175
BC00343=237131,737545,1075175
BC00344=237131,737545,1075175
BC00345=237131,737545,1075175
BC00346=294635,727643,1075175
BC00347=294635,727643,1075175
BC00348=294635,727643,1075175
BC00349=294635,727643,1075175
BC00350=294635,727643,1075175
BC00351=294635,727643,1075175
BC00352=294635,727643,1075175
BC00353=294635,727643,1075175
BC00354=294635,727643,1075175
BC00355=294635,727643,1075175
BC00356=217651,732700,1075175
BC00357=219347,737901,1075175
BC00358=220025,739981,1075175
BC00359=287170,728397,1075175
BC00360=286492,726316,1075175
BC00361=284797,721115,1075175
BC00362=104549,756414,1075175
BC00363=104877,761851,1075175
BC00364=105009,764026,1075175
BC00365=37863,775610,1075175
BC00366=37732,773435,1075175
BC00367=37403,767998,1075175
BC00368=32590,750193,986570
BC00369=32590,674533,986570
BC00370=97174,666880,426359
BC00371=147937,670008,53
BC00372=147937,711773,53
BC00373=147937,730150,53
BC00374=147937,730150,53
BC00375=147937,730150,53
BC00376=147937,730150,53
BC00377=147937,730150,53
BC00378=147937,730150,53
BC00379=147937,730150,53
BC00380=147937,730150,53
BC00381=147937,730150,53
BC00382=147937,730150,53
BC00383=158165,726651,59010
BC00384=158165,726651,59010
BC00385=158165,726651,59010
BC00386=158165,726651,59010
BC00387=158165,726651,59010
BC00388=158165,726651,59010
BC00389=158165,726651,59010
BC00390=158165,726651,59010
BC00391=158165,726651,59010
BC00392=158165,726651,59010
BC00393=154158,704461,35913
BC00394=147937,670008,53
BC00395=303968,673866,53
BC00396=303968,733345,53
BC00397=303968,733345,53
BC00398=303968,733345,53
BC00399=303968,733345,53
BC00400=303968,733345,53
BC00401=303968,733345,53
BC00402=303968,733345,53
BC00403=303968,733345,53
BC00404=303968,733345,53
BC00405=303968,733345,53
BC00406=303968,733345,53
BC00407=303968,733345,53
BC00408=317859,731237,70095
BC00409=317859,731237,70095
BC00410=317859,731237,70095
BC00411=317859,731237,70095
BC00412=317859,731237,70095
BC00413=317859,731237,70095
BC00414=317859,731237,70095
BC00415=317859,731237,70095
BC00416=317859,731237,70095
BC00417=317859,731237,70095
BC00418=294346,742753,94560
BC00419=294346,742753,94560
BC00420=294346,742753,94560
BC00421=294346,742753,94560
BC00422=294346,742753,94560
BC00423=294346,742753,94560
BC00424=294346,742753,94560
BC00425=294346,742753,94560
BC00426=294346,742753,94560
BC00427=294346,742753,94560
BC00428=276740,698523,17248
BC00429=278435,703724,53
BC00430=279113,705804,53
BC00431=283819,705005,53
BC00432=316764,693534,53
BC00433=316086,691453,53
BC00434=314391,686252,53
BC00435=314391,686252,53
BC00436=303968,673866,53
BC00437=147937,670008,53
BC00438=154158,704461,35913
BC00439=166916,707890,15720
BC00440=176272,710404,912
BC00441=176601,715841,53
BC00442=176732,718016,53
BC00443=127735,726480,51
BC00444=162022,730813,53
BC00445=163238,728692,53
BC00446=166278,723391,53
BC00447=166916,707890,15720
BC00448=154158,704461,35913
BC00449=147937,670008,53
BC00450=303968,673866,53
BC00451=314391,686252,53
BC00452=265210,708896,0
BC00453=266905,714097,0
BC00454=267584,716178,0
BC00455=283264,713482,0
BC00456=289747,755484,0
BC00457=287471,755837,0
BC00458=281210,753020,0
BC00459=281210,753020,0
BC00460=281210,753020,0
BC00461=281210,753020,0
BC00462=97174,666880,426359
BC00463=32590,674533,986570
EC00000=-798156,1112951
EC00001=-798156,1112951
EC00002=-798156,1112951
EC00003=-798156,1112951
EC00004=-798156,1112951
EC00005=-798156,1112951
EC00006=-798156,1112951
EC00007=-798156,1112951
EC00008=-798156,1112951
EC00009=-798156,1112951
EC00010=-798156,1112951
EC00011=-798156,1112951
EC00012=-798156,1112951
EC00013=-798156,1112951
EC00014=-798156,1112951
EC00015=-798156,1112951
EC00016=-798156,1112951
EC00017=-798156,1112951
EC00018=-798156,1112951
EC00019=-798156,1112951
EC00020=-798156,1112951
EC00021=-798156,1112951
EC00022=-798156,1112951
EC00023=-798156,1112951
EC00024=-798156,1112951
EC00025=-798153,1112952
EC00026=-798153,1112952
EC00027=-798153,1112952
EC00028=-798153,1112952
EC00029=-798153,1112952
EC00030=-798153,1112952
EC00031=-798153,1112952
EC00032=-798153,1112952
EC00033=-798153,1112952
EC00034=-798153,1112952
EC00035=-798153,1112952
EC00036=-798153,1112952
EC00037=-798153,1112952
EC00038=-798153,1112952
EC00039=-798153,1112952
EC00040=-798153,1112952
EC00041=-798153,1112952
EC00042=-798153,1112952
EC00043=-798153,1112952
EC00044=-798152,1112953
EC00045=-798152,1112953
EC00046=-798152,1112953
EC00047=-798152,1112953
EC00048=-798152,1112953
EC00049=-798152,1112953
EC00050=-798152,1112953
EC00051=-798152,1112953
EC00052=-798152,1112953
EC00053=-798153,1112952
EC00054=-798153,1112952
EC00055=-798153,1112952
EC00056=-798153,1112952
EC00057=-798153,1112952
EC00058=-798153,1112952
EC00059=-798153,1112952
EC00060=-798153,1112952
EC00061=-798153,1112952
EC00062=-798153,1112952
EC00063=-798153,1112952
EC00064=-798153,1112952
EC00065=-798153,1112952
EC00066=-798153,1112952
EC00067=-798153,1112952
EC00068=-798153,1112952
EC00069=-798153,1112952
EC00070=-798153,1112952
EC00071=-798153,1112952
EC00072=-798152,1112952
EC00073=-798152,1112952
EC00074=-798152,1112953
EC00075=-798152,1112953
EC00076=-798151,1112953
EC00077=-798150,1112954
EC00078=-798150,1112954
EC00079=-798150,1112954
EC00080=-798150,1112954
EC00081=-798150,1112954
EC00082=-798150,1112954
EC00083=-798150,1112954
EC00084=-798150,1112954
EC00085=-798150,1112954
EC00086=-798150,1112954
EC00087=-798150,1112954
EC00088=-798150,1112954
EC00089=-798150,1112954
EC00090=-798150,1112954
EC00091=-798150,1112954
EC00092=-798156,1112951
EC00093=-798156,1112951
EC00094=-798156,1112951
EC00095=-798156,1112951
EC00096=-798156,1112951
EC00097=-798156,1112951
EC00098=-798156,1112951
EC00099=-798156,1112951
EC00100=-798156,1112951
EC00101=-798156,1112951
EC00102=-798156,1112951
EC00103=-798156,1112951
EC00104=-798156,1112951
EC00105=-798156,1112951
EC00106=-798156,1112951
EC00107=-798156,1112951
EC00108=-798156,1112951
EC00109=-798156,1112951
EC00110=-798156,1112951
EC00111=-798155,1112952
EC00112=-798156,1112951
EC00113=-798156,1112951
EC00114=-798155,1112952
EC00115=-798156,1112951
EC00116=-798156,1112951
EC00117=-798156,1112951
EC00118=-798156,1112951
EC00119=-798156,1112951
EC00120=-798156,1112951
EC00121=-798156,1112951
EC00122=-798156,1112951
EC00123=-798156,1112951
EC00124=-798156,1112951
EC00125=-798156,1112951
EC00126=-798156,1112951
EC00127=-798156,1112951
EC00128=-798156,1112951
EC00129=-798156,1112951
EC00130=-798156,1112951
EC00131=-798156,1112951
EC00132=-798156,1112951
EC00133=-798156,1112951
EC00134=-798156,1112951
EC00135=-798156,1112951
EC00136=-798156,1112951
EC00137=-798156,1112951
EC00138=-798156,1112951
EC00139=-798156,1112951
EC00140=-798156,1112951
EC00141=-798156,1112951
EC00142=-798156,1112951
EC00143=-798156,1112951
EC00144=-798156,1112951
EC00145=-798156,1112951
EC00146=-798156,1112951
EC00147=-798156,1112951
EC00148=-798156,1112951
EC00149=-798156,1112951
EC00150=-798156,1112951
EC00151=-798156,1112951
EC00152=-798156,1112951
EC00153=-798156,1112951
EC00154=-798156,1112951
EC00155=-798156,1112951
EC00156=-798156,1112951
EC00157=-798156,1112951
EC00158=-798156,1112951
EC00159=-798156,1112951
EC00160=-798156,1112951
EC00161=-798156,1112951
EC00162=-798156,1112951
EC00163=-798156,1112951
EC00164=-798156,1112951
EC00165=-798156,1112951
EC00166=-798156,1112951
EC00167=-798156,1112951
EC00168=-798156,1112951
EC00169=-798156,1112951
EC00170=-798156,1112951
EC00171=-798156,1112951
EC00172=-798153,1112952
EC00173=-798153,1112952
EC00174=-798153,1112952
EC00175=-798152,1112952
EC00176=-798152,1112952
EC00177=-798152,1112952
EC00178=-798152,1112952
EC00179=-798152,1112952
EC00180=-798152,1112952
EC00181=-798152,1112952
EC00182=-798152,1112952
EC00183=-798152,1112952
EC00184=-798152,1112952
EC00185=-798152,1112952
EC00186=-798152,1112952
EC00187=-798151,1112953
EC00188=-798151,1112953
EC00189=-798151,1112953
EC00190=-798151,1112953
EC00191=-798151,1112953
EC00192=-798151,1112953
EC00193=-798151,1112953
EC00194=-798151,1112953
EC00195=-798151,1112953
EC00196=-798151,1112953
EC00197=-798151,1112953
EC00198=-798151,1112953
EC00199=-798151,1112953
EC00200=-798151,1112953
EC00201=-798151,1112953
EC00202=-798151,1112953
EC00203=-798151,1112953
EC00204=-798151,1112953
EC00205=-798151,1112953
EC00206=-798151,1112953
EC00207=-798151,1112953
EC00208=-798151,1112953
EC00209=-798151,1112953
EC00210=-798151,1112953
EC00211=-798151,1112953
EC00212=-798151,1112953
EC00213=-798151,1112953
EC00214=-798151,1112953
EC00215=-798150,1112954
EC00216=-798150,1112954
EC00217=-798150,1112954
EC00218=-798150,1112954
EC00219=-798150,1112954
EC00220=-798150,1112954
EC00221=-798150,1112954
EC00222=-798150,1112954
EC00223=-798150,1112954
EC00224=-798150,1112954
EC00225=-798150,1112954
EC00226=-798150,1112954
EC00227=-798150,1112954
EC00228=-798150,1112954
EC00229=-798150,1112954
EC00230=-798155,1112952
EC00231=-798156,1112951
EC00232=-798156,1112951
EC00233=-798156,1112951
EC00234=-798156,1112951
EC00235=-798156,1112951
EC00236=-798156,1112951
EC00237=-798156,1112951
EC00238=-798156,1112951
EC00239=-798156,1112951
EC00240=-798156,1112951
EC00241=-798156,1112951
EC00242=-798156,1112951
EC00243=-798156,1112951
EC00244=-798156,1112951
EC00245=-798155,1112951
EC00246=-798156,1112951
EC00247=-798156,1112951
EC00248=-798156,1112951
EC00249=-798156,1112951
EC00250=-798156,1112951
EC00251=-798156,1112951
EC00252=-798156,1112951
EC00253=-798156,1112951
EC00254=-798156,1112951
EC00255=-798156,1112951
EC00256=-798156,1112951
EC00257=-798156,1112951
EC00258=-798156,1112951
EC00259=-798156,1112951
EC00260=-798156,1112951
EC00261=-798156,1112951
EC00262=-798156,1112951
EC00263=-798156,1112951
EC00264=-798156,1112951
EC00265=-798156,1112951
EC00266=-798156,1112951
EC00267=-798156,1112951
EC00268=-798156,1112951
EC00269=-798156,1112951
EC00270=-798156,1112951
EC00271=-798156,1112951
EC00272=-798156,1112951
EC00273=-798156,1112951
EC00274=-798156,1112951
EC00275=-798156,1112951
EC00276=-798156,1112951
EC00277=-798156,1112951
EC00278=-798156,1112951
EC00279=-798156,1112951
EC00280=-798156,1112951
EC00281=-798156,1112951
EC00282=-798156,1112951
EC00283=-798156,1112951
EC00284=-798156,1112951
EC00285=-798156,1112951
EC00286=-798156,1112951
EC00287=-798156,1112951
EC00288=-798156,1112951
EC00289=-798156,1112951
EC00290=-798156,1112951
EC00291=-798156,1112951
EC00292=-798156,1112951
EC00293=-798156,1112951
EC00294=-798156,1112951
EC00295=-798156,1112951
EC00296=-798156,1112951
EC00297=-798156,1112951
EC00298=-798156,1112951
EC00299=-798156,1112951
EC00300=-798156,1112951
EC00301=-798156,1112951
EC00302=-798156,1112951
EC00303=-798156,1112951
EC00304=-798156,1112951
EC00305=-798156,1112951
EC00306=-798155,1112951
EC00307=-798156,1112951
EC00308=-798156,1112951
EC00309=-798156,1112951
EC00310=-798156,1112951
EC00311=-850885,799301
EC00312=-850885,361850
EC00313=-798154,-3
EC00314=-798156,0
EC00315=-798156,0
EC00316=-798156,0
EC00317=-798156,0
EC00318=-798156,0
EC00319=-798156,0
EC00320=-798156,0
EC00321=-798156,0
EC00322=-798156,0
EC00323=-798156,0
EC00324=-798156,0
EC00325=-798156,0
EC00326=-798156,0
EC00327=-798156,0
EC00328=-798156,0
EC00329=-798156,0
EC00330=-798156,0
EC00331=-798156,0
EC00332=-798156,0
EC00333=-798156,0
EC00334=-798156,0
EC00335=-798156,0
EC00336=-798156,0
EC00337=-798156,0
EC00338=-798156,0
EC00339=-798156,0
EC00340=-798156,0
EC00341=-798156,0
EC00342=-798156,0
EC00343=-798156,0
EC00344=-798156,0
EC00345=-798156,0
EC00346=-798156,0
EC00347=-798156,0
EC00348=-798156,0
EC00349=-798156,0
EC00350=-798156,0
EC00351=-798156,0
EC00352=-798156,0
EC00353=-798156,0
EC00354=-798156,0
EC00355=-798156,0
EC00356=-798156,0
EC00357=-798156,0
EC00358=-798156,0
EC00359=-798156,0
EC00360=-798156,0
EC00361=-798156,0
EC00362=-798156,0
EC00363=-798156,0
EC00364=-798156,0
EC00365=-798156,0
EC00366=-798156,0
EC00367=-798156,0
EC00368=-798156,0
EC00369=-798156,0
EC00370=-798156,0
EC00371=-798156,0
EC00372=-798156,0
EC00373=-798156,0
EC00374=-798156,0
EC00375=-798156,0
EC00376=-798156,0
EC00377=-798156,0
EC00378=-798156,0
EC00379=-798156,0
EC00380=-798156,0
EC00381=-798156,0
EC00382=-798156,0
EC00383=-798156,0
EC00384=-798156,0
EC00385=-798156,0
EC00386=-798156,0
EC00387=-798156,0
EC00388=-798156,0
EC00389=-798156,0
EC00390=-798156,0
EC00391=-798156,0
EC00392=-798156,0
EC00393=-798156,0
EC00394=-798156,0
EC00395=-798156,0
EC00396=-798156,0
EC00397=-798156,0
EC00398=-798156,0
EC00399=-798156,0
EC00400=-798156,0
EC00401=-798156,0
EC00402=-798156,0
EC00403=-798156,0
EC00404=-798156,0
EC00405=-798156,0
EC00406=-798156,0
EC00407=-798156,0
EC00408=-798156,0
EC00409=-798156,0
EC00410=-798156,0
EC00411=-798156,0
EC00412=-798156,0
EC00413=-798156,0
EC00414=-798156,0
EC00415=-798156,0
EC00416=-798156,0
EC00417=-798156,0
EC00418=-798156,0
EC00419=-798156,0
EC00420=-798156,0
EC00421=-798156,0
EC00422=-798156,0
EC00423=-798156,0
EC00424=-798156,0
EC00425=-798156,0
EC00426=-798156,0
EC00427=-798156,0
EC00428=-798156,0
EC00429=-798156,0
EC00430=-798156,0
EC00431=-798156,0
EC00432=-798156,0
EC00433=-798156,0
EC00434=-798156,0
EC00435=-798156,0
EC00436=-798156,0
EC00437=-798156,0
EC00438=-798156,0
EC00439=-798156,0
EC00440=-798156,0
EC00441=-798156,0
EC00442=-798156,0
EC00443=-798155,-1
EC00444=-798156,0
EC00445=-798156,0
EC00446=-798156,0
EC00447=-798156,0
EC00448=-798156,0
EC00449=-798156,0
EC00450=-798156,0
EC00451=-798156,0
EC00452=-798156,0
EC00453=-798156,0
EC00454=-798156,0
EC00455=-798156,0
EC00456=-798156,0
EC00457=-798156,0
EC00458=-798156,0
EC00459=-798156,0
EC00460=-798156,0
EC00461=-798156,0
EC00462=-798156,0
EC00463=-798156,0
///POSTYPE BASE
///RECTAN
///RCONF 0,0,0,0,0,0,0,0,0,0,0,0,0,0,0,0,0,0,0,0,0,0,0,0
P00006=0.222,-3.123,-1.508,0.0000,0.0000,0.0000
P00021=-0.225,-6.128,-0.405,0.0000,0.0000,0.0000
P00022=0.222,-3.123,-1.508,0.0000,0.0000,0.0000
P00023=0.143,-0.036,0.682,0.0000,0.0000,0.0000
P00024=0.145,-0.552,1.326,0.0000,0.0000,0.0000
P00025=-2.003,0.006,0.728,0.0000,0.0000,0.0000
P00026=0.562,-0.002,-0.337,0.0000,0.0000,0.0000
P00027=-0.746,0.015,-9.096,0.0000,0.0000,0.0000
P00028=-2.237,-0.018,-7.702,0.0000,0.0000,0.0000
///RCONF 0,0,0,0,1,0,0,0,0,0,0,0,0,0,0,0,0,0,0,0,0,0,0,0
P00033=-0.123,0.612,-5.012,0.0000,0.0000,0.0000
///RCONF 0,0,0,0,0,0,0,0,0,0,0,0,0,0,0,0,0,0,0,0,0,0,0,0
P00034=-0.304,0.773,-2.693,0.0000,0.0000,0.0000
P00035=2.817,0.591,-1.622,0.0000,0.0000,0.0000
P00036=-1.108,-0.829,1.850,0.0000,0.0000,0.0000
P00041=0.192,3.924,0.305,0.0000,0.0000,0.0000
P00042=-0.217,1.941,0.413,0.0000,0.0000,0.0000
P00043=-0.044,-1.937,1.197,0.0000,0.0000,0.0000
P00044=0.687,-2.322,1.156,0.0000,0.0000,0.0000
P00045=-0.068,-0.810,1.603,0.0000,0.0000,0.0000
P00046=0.799,0.043,1.292,0.0000,0.0000,0.0000
P00051=0.367,3.892,0.009,0.0000,0.0000,0.0000
P00052=0.088,2.832,-0.342,0.0000,0.0000,0.0000
P00053=0.134,6.594,0.107,0.0000,0.0000,0.0000
P00054=-0.103,6.509,-0.702,0.0000,0.0000,0.0000
P00055=-0.342,8.912,1.324,0.0000,0.0000,0.0000
P00056=0.568,-0.032,0.830,0.0000,0.0000,0.0000
P00057=0.586,-0.180,1.727,0.0000,0.0000,0.0000
P00058=0.385,-0.061,1.027,0.0000,0.0000,0.0000
P00059=0.483,-0.984,-2.888,0.0000,0.0000,0.0000
P00060=2.327,-2.514,-2.692,0.0000,0.0000,0.0000
P00061=1.575,-3.405,-0.752,0.0000,0.0000,0.0000
//INST
///DATE 2025/03/12 15:15
///ATTR SC,RW
///GROUP1 RB1,BS1
///GROUP2 ST1
NOP
'X2_29-32(-90,180)
MOVJ C00000 BC00000 VJ=100.00  +MOVJ EC00000 VJ=100.00
MOVJ C00001 BC00001 VJ=100.00  +MOVJ EC00001 VJ=100.00
MOVJ C00002 BC00002 VJ=100.00  +MOVJ EC00002 VJ=100.00
MOVJ C00003 BC00003 VJ=100.00  +MOVJ EC00003 VJ=100.00
MOVJ C00004 BC00004 VJ=100.00  +MOVJ EC00004 VJ=100.00
'Path S4862
SFTOF3D
MOVJ C00005 BC00005 VJ=100.00  +MOVJ EC00005 VJ=100.00
MOVL C00006 BC00006 V=800.0  +MOVJ EC00006 VJ=100.00
SMOVL C00007 BC00007 V=166.7  +MOVJ EC00007
SREFP 3 C00008 BC00008  +REFP EC00008
CALL JOB:SEARCH-R1-S13D
SET P042 P006
SFTON3D P042
SMOVL C00009 BC00009 V=166.7  +MOVJ EC00009
SMOVL C00010 BC00010 V=166.7  +MOVJ EC00010
SREFP 3 C00011 BC00011  +REFP EC00011
CALL JOB:SEARCH-R1-S13D
SET P042 P006
SFTON3D P042
SMOVL C00012 BC00012 V=166.7  +MOVJ EC00012
MOVL C00013 BC00013 V=800.0  +MOVJ EC00013 VJ=100.00
MOVL C00014 BC00014 V=1000.0  +MOVJ EC00014 VJ=100.00
'EndPath S4862
'Path S4863
SFTOF3D
MOVJ C00015 BC00015 VJ=100.00  +MOVJ EC00015 VJ=100.00
MOVL C00016 BC00016 V=800.0  +MOVJ EC00016 VJ=100.00
SMOVL C00017 BC00017 V=166.7  +MOVJ EC00017
SREFP 3 C00018 BC00018  +REFP EC00018
CALL JOB:SEARCH-R1-S13D
SET P041 P006
SFTON3D P041
SMOVL C00019 BC00019 V=166.7  +MOVJ EC00019
SMOVL C00020 BC00020 V=166.7  +MOVJ EC00020
SREFP 3 C00021 BC00021  +REFP EC00021
CALL JOB:SEARCH-R1-S13D
SET P041 P006
SFTON3D P041
SMOVL C00022 BC00022 V=166.7  +MOVJ EC00022
MOVL C00023 BC00023 V=800.0  +MOVJ EC00023 VJ=100.00
MOVL C00024 BC00024 V=1000.0  +MOVJ EC00024 VJ=100.00
SFTOF3D
MOVJ C00025 BC00025 VJ=30.00  +MOVJ EC00025 VJ=30.00
MOVJ C00026 BC00026 VJ=30.00  +MOVJ EC00026 VJ=100.00
SMOVL C00027 BC00027 V=166.7  +MOVJ EC00027
SREFP 3 C00028 BC00028  +REFP EC00028
CALL JOB:SEARCH-R1-S13D
SET P051 P006
SFTON3D P051
SMOVL C00029 BC00029 V=166.7  +MOVJ EC00029
SREFP 3 C00030 BC00030  +REFP EC00030
CALL JOB:SEARCH-R1-S13D
SET P051 P006
SFTON3D P051
SMOVL C00031 BC00031 V=166.7  +MOVJ EC00031
SMOVL C00032 BC00032 V=166.7  +MOVJ EC00032
SREFP 3 C00033 BC00033  +REFP EC00033
CALL JOB:SEARCH-R1-S13D
SET P051 P006
SFTON3D P051
SMOVL C00034 BC00034 V=166.7  +MOVJ EC00034
SMOVL C00035 BC00035 V=166.7  +MOVJ EC00035
SREFP 3 C00036 BC00036  +REFP EC00036
CALL JOB:SEARCH-R1-S13D
SET P052 P006
SFTON3D P052
SMOVL C00037 BC00037 V=166.7  +MOVJ EC00037
SREFP 3 C00038 BC00038  +REFP EC00038
CALL JOB:SEARCH-R1-S13D
SET P052 P006
SFTON3D P052
SMOVL C00039 BC00039 V=166.7  +MOVJ EC00039
SREFP 3 C00040 BC00040  +REFP EC00040
CALL JOB:SEARCH-R1-S13D
SET P052 P006
SFTON3D P052
SMOVL C00041 BC00041 V=166.7  +MOVJ EC00041
MOVL C00042 BC00042 V=1000.0  +MOVJ EC00042 VJ=30.00
SMOVL C00043 BC00043 V=166.7 PL=0  +MOVJ EC00043
SREFP 3 C00044 BC00044  +REFP EC00044
CALL JOB:SEARCH-R1-S13D
SET P053 P006
SFTON3D P053
SMOVL C00045 BC00045 V=166.7  +MOVJ EC00045
SREFP 3 C00046 BC00046  +REFP EC00046
CALL JOB:SEARCH-R1-S13D
SET P053 P006
SFTON3D P053
SMOVL C00047 BC00047 V=166.7  +MOVJ EC00047
SMOVL C00048 BC00048 V=166.7 PL=0  +MOVJ EC00048
SREFP 3 C00049 BC00049  +REFP EC00049
CALL JOB:SEARCH-R1-S13D
SET P054 P006
SFTON3D P054
SMOVL C00050 BC00050 V=166.7  +MOVJ EC00050
SREFP 3 C00051 BC00051  +REFP EC00051
CALL JOB:SEARCH-R1-S13D
SET P054 P006
SFTON3D P054
SMOVL C00052 BC00052 V=166.7  +MOVJ EC00052
SFTOF3D
SMOVL C00053 BC00053 V=1000.0  +MOVJ EC00053
SMOVL C00054 BC00054 V=1000.0  +MOVJ EC00054
SMOVL C00055 BC00055 V=1000.0  +MOVJ EC00055
SMOVL C00056 BC00056 V=166.7  +MOVJ EC00056
SREFP 3 C00057 BC00057  +REFP EC00057
CALL JOB:SEARCH-R1-S13D
SET P055 P006
SFTON3D P055
SMOVL C00058 BC00058 V=166.7  +MOVJ EC00058
SREFP 3 C00059 BC00059  +REFP EC00059
CALL JOB:SEARCH-R1-S13D
SET P055 P006
SFTON3D P055
SMOVL C00060 BC00060 V=166.7  +MOVJ EC00060
SMOVL C00061 BC00061 V=166.7  +MOVJ EC00061
SREFP 3 C00062 BC00062  +REFP EC00062
CALL JOB:SEARCH-R1-S13D
SET P055 P006
SFTON3D P055
SMOVL C00063 BC00063 V=166.7  +MOVJ EC00063
SMOVL C00064 BC00064 V=166.7  +MOVJ EC00064
SREFP 3 C00065 BC00065  +REFP EC00065
CALL JOB:SEARCH-R1-S13D
SET P056 P006
SFTON3D P056
SMOVL C00066 BC00066 V=166.7  +MOVJ EC00066
SREFP 3 C00067 BC00067  +REFP EC00067
CALL JOB:SEARCH-R1-S13D
SET P056 P006
SFTON3D P056
SMOVL C00068 BC00068 V=166.7  +MOVJ EC00068
SMOVL C00069 BC00069 V=166.7  +MOVJ EC00069
SREFP 3 C00070 BC00070  +REFP EC00070
CALL JOB:SEARCH-R1-S13D
SET P056 P006
SFTON3D P056
SMOVL C00071 BC00071 V=166.7  +MOVJ EC00071
SFTOF3D
SMOVL C00072 BC00072 V=1000.0  +MOVJ EC00072
SMOVL C00073 BC00073 V=1000.0  +MOVJ EC00073
SMOVL C00074 BC00074 V=1000.0  +MOVJ EC00074
SMOVL C00075 BC00075 V=166.7 PL=0  +MOVJ EC00075
SREFP 3 C00076 BC00076  +REFP EC00076
CALL JOB:SEARCH-R1-S13D
SET P057 P006
SFTON3D P057
SMOVL C00077 BC00077 V=166.7  +MOVJ EC00077
SREFP 3 C00078 BC00078  +REFP EC00078
CALL JOB:SEARCH-R1-S13D
SET P057 P006
SFTON3D P057
SMOVL C00079 BC00079 V=166.7  +MOVJ EC00079
SMOVL C00080 BC00080 V=166.7  +MOVJ EC00080
SREFP 3 C00081 BC00081  +REFP EC00081
CALL JOB:SEARCH-R1-S13D
SET P058 P006
SFTON3D P058
SMOVL C00082 BC00082 V=166.7  +MOVJ EC00082
SREFP 3 C00083 BC00083  +REFP EC00083
CALL JOB:SEARCH-R1-S13D
SET P058 P006
SFTON3D P058
SMOVL C00084 BC00084 V=166.7  +MOVJ EC00084
SMOVL C00085 BC00085 V=166.7  +MOVJ EC00085
SMOVL C00086 BC00086 V=166.7 PL=0  +MOVJ EC00086
SREFP 3 C00087 BC00087  +REFP EC00087
CALL JOB:SEARCH-R1-S13D
SET P059 P006
SFTON3D P059
SMOVL C00088 BC00088 V=166.7  +MOVJ EC00088
SREFP 3 C00089 BC00089  +REFP EC00089
CALL JOB:SEARCH-R1-S13D
SET P059 P006
SFTON3D P059
SMOVL C00090 BC00090 V=166.7  +MOVJ EC00090
SFTOF3D
SMOVL C00091 BC00091 V=666.7  +MOVJ EC00091
'EndPath S4863
MOVJ C00092 BC00092 VJ=100.00  +MOVJ EC00092 VJ=100.00
MOVJ C00093 BC00093 VJ=100.00  +MOVJ EC00093 VJ=100.00
MOVJ C00094 BC00094 VJ=100.00  +MOVJ EC00094 VJ=100.00
MOVJ C00095 BC00095 VJ=100.00  +MOVJ EC00095 VJ=100.00
MOVJ C00096 BC00096 VJ=30.00  +MOVJ EC00096 VJ=30.00
MOVJ C00097 BC00097 VJ=30.00  +MOVJ EC00097 VJ=30.00
MOVL C00098 BC00098 V=166.7  +MOVJ EC00098 VJ=0.78
SMOVL C00099 BC00099 V=166.7  +MOVJ EC00099
SREFP 3 C00100 BC00100  +REFP EC00100
CALL JOB:SEARCH-R1-S13D
SET P060 P006
SFTON3D P060
SMOVL C00101 BC00101 V=166.7  +MOVJ EC00101
SREFP 3 C00102 BC00102  +REFP EC00102
CALL JOB:SEARCH-R1-S13D
SET P060 P006
SFTON3D P060
SMOVL C00103 BC00103 V=166.7  +MOVJ EC00103
SMOVL C00104 BC00104 V=166.7  +MOVJ EC00104
SREFP 3 C00105 BC00105  +REFP EC00105
CALL JOB:SEARCH-R1-S13D
SET P060 P006
SFTON3D P060
SMOVL C00106 BC00106 V=166.7  +MOVJ EC00106
SMOVL C00107 BC00107 V=166.7  +MOVJ EC00107
SREFP 3 C00108 BC00108  +REFP EC00108
CALL JOB:SEARCH-R1-S13D
SET P061 P006
SFTON3D P061
SMOVL C00109 BC00109 V=166.7  +MOVJ EC00109
SREFP 3 C00110 BC00110  +REFP EC00110
CALL JOB:SEARCH-R1-S13D
SET P061 P006
SFTON3D P061
SMOVL C00111 BC00111 V=166.7  +MOVJ EC00111
SMOVL C00112 BC00112 V=166.7  +MOVJ EC00112
SREFP 3 C00113 BC00113  +REFP EC00113
CALL JOB:SEARCH-R1-S13D
SET P061 P006
SFTON3D P061
SMOVL C00114 BC00114 V=166.7  +MOVJ EC00114
SFTOF3D
MOVL C00115 BC00115 V=166.7  +MOVJ EC00115 VJ=0.78
MOVJ C00116 BC00116 VJ=30.00  +MOVJ EC00116 VJ=30.00
'Path S4864
SFTOF3D
MOVJ C00117 BC00117 VJ=100.00  +MOVJ EC00117 VJ=100.00
MOVL C00118 BC00118 V=800.0  +MOVJ EC00118 VJ=100.00
SMOVL C00119 BC00119 V=166.7  +MOVJ EC00119
SREFP 3 C00120 BC00120  +REFP EC00120
CALL JOB:SEARCH-R1-S13D
SET P045 P006
SFTON3D P045
SMOVL C00121 BC00121 V=166.7  +MOVJ EC00121
SREFP 3 C00122 BC00122  +REFP EC00122
CALL JOB:SEARCH-R1-S13D
SET P045 P006
SFTON3D P045
SMOVL C00123 BC00123 V=166.7  +MOVJ EC00123
MOVL C00124 BC00124 V=800.0  +MOVJ EC00124 VJ=100.00
MOVL C00125 BC00125 V=1000.0  +MOVJ EC00125 VJ=100.00
'EndPath S4864
'Path S4231
SFTOF3D
MOVJ C00126 BC00126 VJ=100.00  +MOVJ EC00126 VJ=100.00
MOVL C00127 BC00127 V=800.0  +MOVJ EC00127 VJ=100.00
SMOVL C00128 BC00128 V=166.7  +MOVJ EC00128
SREFP 3 C00129 BC00129  +REFP EC00129
CALL JOB:SEARCH-R1-S13D
SET P022 P006
SFTON3D P022
SMOVL C00130 BC00130 V=166.7  +MOVJ EC00130
SREFP 3 C00131 BC00131  +REFP EC00131
CALL JOB:SEARCH-R1-S13D
SET P022 P006
SFTON3D P022
SMOVL C00132 BC00132 V=166.7  +MOVJ EC00132
MOVL C00133 BC00133 V=800.0  +MOVJ EC00133 VJ=100.00
MOVL C00134 BC00134 V=1000.0  +MOVJ EC00134 VJ=100.00
'EndPath S4231
'Path S4232
SFTOF3D
MOVJ C00135 BC00135 VJ=100.00  +MOVJ EC00135 VJ=100.00
MOVL C00136 BC00136 V=800.0  +MOVJ EC00136 VJ=100.00
SMOVL C00137 BC00137 V=166.7  +MOVJ EC00137
SREFP 3 C00138 BC00138  +REFP EC00138
CALL JOB:SEARCH-R1-S13D
SET P021 P006
SFTON3D P021
SMOVL C00139 BC00139 V=166.7  +MOVJ EC00139
SREFP 3 C00140 BC00140  +REFP EC00140
CALL JOB:SEARCH-R1-S13D
SET P021 P006
SFTON3D P021
SMOVL C00141 BC00141 V=166.7  +MOVJ EC00141
MOVL C00142 BC00142 V=800.0  +MOVJ EC00142 VJ=100.00
MOVL C00143 BC00143 V=1000.0  +MOVJ EC00143 VJ=100.00
'EndPath S4232
'Path W4886
SFTOF3D
SFTON3D P021
MOVJ C00144 BC00144 VJ=100.00  +MOVJ EC00144 VJ=100.00
SMOVL C00145 BC00145 V=800.0  +MOVJ EC00145
SMOVL C00146 BC00146 V=150.0 PL=0  +MOVJ EC00146
MACRO1 MJ#(0) ARGF6
ARCON
SMOVL C00147 BC00147 V=8.3  +MOVJ EC00147
SFTON3D P022
SMOVL C00148 BC00148 V=8.3  +MOVJ EC00148
ARCOF
SMOVL C00149 BC00149 V=800.0  +MOVJ EC00149
SMOVL C00150 BC00150 V=1000.0  +MOVJ EC00150
SFTOF3D
'EndPath W4886
MOVJ C00151 BC00151 VJ=100.00  +MOVJ EC00151 VJ=100.00
MOVJ C00152 BC00152 VJ=30.00  +MOVJ EC00152 VJ=30.00
MOVJ C00153 BC00153 VJ=30.00  +MOVJ EC00153 VJ=30.00
MOVL C00154 BC00154 V=166.7  +MOVJ EC00154 VJ=0.78
SFTON3D P060
SMOVL C00155 BC00155 V=166.7  +MOVJ EC00155
SMOVL C00156 BC00156 V=150.0 PL=0  +MOVJ EC00156
MACRO1 MJ#(0) ARGF9
ARCON
SFTON3D P061
SMOVL C00157 BC00157 V=10.0  +MOVJ EC00157
SMOVC C00158 BC00158 V=13.3  +MOVJ EC00158
SMOVC C00159 BC00159 V=13.3  +MOVJ EC00159
SMOVC C00160 BC00160 V=13.3  +MOVJ EC00160
SFTON3D P060
SMOVL C00161 BC00161 V=10.0  +MOVJ EC00161
SMOVL C00162 BC00162 V=10.0  +MOVJ EC00162
SMOVC C00163 BC00163 V=13.3  +MOVJ EC00163
SMOVC C00164 BC00164 V=13.3  +MOVJ EC00164
SMOVC C00165 BC00165 V=13.3  +MOVJ EC00165
ARCOF
SMOVL C00166 BC00166 V=166.7  +MOVJ EC00166
SFTOF3D
SMOVL C00167 BC00167 V=666.7  +MOVJ EC00167
MOVJ C00168 BC00168 VJ=100.00  +MOVJ EC00168 VJ=0.78
MOVJ C00169 BC00169 VJ=100.00  +MOVJ EC00169 VJ=100.00
MOVJ C00170 BC00170 VJ=100.00  +MOVJ EC00170 VJ=100.00
MOVJ C00171 BC00171 VJ=100.00  +MOVJ EC00171 VJ=100.00
MOVJ C00172 BC00172 VJ=100.00  +MOVJ EC00172 VJ=100.00
MOVJ C00173 BC00173 VJ=100.00  +MOVJ EC00173 VJ=100.00
SFTON3D P055
MOVJ C00174 BC00174 VJ=50.00  +MOVJ EC00174 VJ=100.00
SMOVL C00175 BC00175 V=150.0 PL=0  +MOVJ EC00175
MACRO1 MJ#(0) ARGF9
ARCON
SFTON3D P056
SMOVL C00176 BC00176 V=10.0  +MOVJ EC00176
SMOVC C00177 BC00177 V=13.3  +MOVJ EC00177
SMOVC C00178 BC00178 V=13.3  +MOVJ EC00178
SMOVC C00179 BC00179 V=13.3  +MOVJ EC00179
SFTON3D P055
SMOVL C00180 BC00180 V=10.0  +MOVJ EC00180
SMOVL C00181 BC00181 V=10.0  +MOVJ EC00181
SMOVC C00182 BC00182 V=13.3  +MOVJ EC00182
SMOVC C00183 BC00183 V=13.3  +MOVJ EC00183
SMOVC C00184 BC00184 V=13.3  +MOVJ EC00184
ARCOF
SMOVL C00185 BC00185 V=166.7  +MOVJ EC00185
SFTOF3D
MOVL C00186 BC00186 V=166.7  +MOVJ EC00186 VJ=0.78
SFTON3D P051
SMOVL C00187 BC00187 V=150.0 PL=0  +MOVJ EC00187
MACRO1 MJ#(0) ARGF9
ARCON
SFTON3D P052
SMOVL C00188 BC00188 V=10.0  +MOVJ EC00188
SMOVC C00189 BC00189 V=13.3  +MOVJ EC00189
SMOVC C00190 BC00190 V=13.3  +MOVJ EC00190
SMOVC C00191 BC00191 V=13.3  +MOVJ EC00191
SFTON3D P051
SMOVL C00192 BC00192 V=10.0  +MOVJ EC00192
SMOVL C00193 BC00193 V=10.0  +MOVJ EC00193
SMOVC C00194 BC00194 V=13.3  +MOVJ EC00194
SMOVC C00195 BC00195 V=13.3  +MOVJ EC00195
SMOVC C00196 BC00196 V=13.3  +MOVJ EC00196
ARCOF
SMOVL C00197 BC00197 V=166.7  +MOVJ EC00197
SFTOF3D
MOVJ C00198 BC00198 VJ=100.00  +MOVJ EC00198 VJ=0.78
MOVL C00199 BC00199 V=333.3  +MOVJ EC00199 VJ=100.00
SFTON3D P057
MOVL C00200 BC00200 V=333.3  +MOVJ EC00200 VJ=100.00
SMOVL C00201 BC00201 V=83.3  +MOVJ EC00201
ARCON
SMOVL C00202 BC00202 V=10.0  +MOVJ EC00202
SMOVC C00203 BC00203 V=13.3  +MOVJ EC00203
SMOVC C00204 BC00204 V=13.3  +MOVJ EC00204
SMOVC C00205 BC00205 V=13.3  +MOVJ EC00205
SMOVC C00206 BC00206 V=13.3  +MOVJ EC00206
SFTON3D P058
SMOVL C00207 BC00207 V=10.0  +MOVJ EC00207
SMOVC C00208 BC00208 V=13.3  +MOVJ EC00208
SFTON3D P059
SMOVC C00209 BC00209 V=13.3  +MOVJ EC00209
SMOVC C00210 BC00210 V=13.3  +MOVJ EC00210
SMOVL C00211 BC00211 V=10.0  +MOVJ EC00211
ARCOF
SMOVL C00212 BC00212 V=166.7  +MOVJ EC00212
SFTOF3D
SMOVL C00213 BC00213 V=666.7  +MOVJ EC00213
SMOVL C00214 BC00214 V=666.7  +MOVJ EC00214
SMOVL C00215 BC00215 V=666.7  +MOVJ EC00215
SMOVL C00216 BC00216 V=666.7  +MOVJ EC00216
SFTON3D P053
SMOVL C00217 BC00217 V=166.7 PL=0  +MOVJ EC00217
ARCON
SWVON WEV#(70)
SMOVL C00218 BC00218 V=6.7  +MOVJ EC00218
ARCOF
SWVOF
SMOVL C00219 BC00219 V=166.7  +MOVJ EC00219
SMOVL C00220 BC00220 V=83.3  +MOVJ EC00220
SMOVL C00221 BC00221 V=83.3  +MOVJ EC00221
ARCON
SWVON WEV#(70)
SMOVL C00222 BC00222 V=6.7  +MOVJ EC00222
SFTON3D P054
SMOVL C00223 BC00223 V=6.7  +MOVJ EC00223
ARCOF
SWVOF
SMOVL C00224 BC00224 V=166.7  +MOVJ EC00224
SMOVL C00225 BC00225 V=166.7  +MOVJ EC00225
SMOVL C00226 BC00226 V=83.3  +MOVJ EC00226
ARCON
SWVON WEV#(70)
SMOVL C00227 BC00227 V=6.7  +MOVJ EC00227
ARCOF
SWVOF
SMOVL C00228 BC00228 V=333.3  +MOVJ EC00228
SFTOF3D
SMOVL C00229 BC00229 V=333.3  +MOVJ EC00229
SMOVL C00230 BC00230 V=666.7  +MOVJ EC00230
'Path W4887
SFTOF3D
SFTON3D P041
MOVJ C00231 BC00231 VJ=100.00  +MOVJ EC00231 VJ=100.00
SMOVL C00232 BC00232 V=800.0  +MOVJ EC00232
MACRO1 MJ#(0) ARGF6
SMOVL C00233 BC00233 V=150.0 PL=0  +MOVJ EC00233
ARCON
SMOVL C00234 BC00234 V=8.3  +MOVJ EC00234
SFTON3D P042
SMOVL C00235 BC00235 V=8.3  +MOVJ EC00235
ARCOF
SMOVL C00236 BC00236 V=800.0  +MOVJ EC00236
SMOVL C00237 BC00237 V=1000.0  +MOVJ EC00237
SFTOF3D
'EndPath W4887
MOVJ C00238 BC00238 VJ=100.00  +MOVJ EC00238 VJ=100.00
MOVJ C00239 BC00239 VJ=100.00  +MOVJ EC00239 VJ=100.00
MOVJ C00240 BC00240 VJ=100.00  +MOVJ EC00240 VJ=100.00
MOVJ C00241 BC00241 VJ=100.00  +MOVJ EC00241 VJ=100.00
MOVJ C00242 BC00242 VJ=100.00  +MOVJ EC00242 VJ=100.00
'Path W4887
SFTOF3D
SFTON3D P045
MOVJ C00243 BC00243 VJ=100.00  +MOVJ EC00243 VJ=100.00
SMOVL C00244 BC00244 V=800.0  +MOVJ EC00244
SMOVL C00245 BC00245 V=150.0 PL=0  +MOVJ EC00245
ARCON
SMOVL C00246 BC00246 V=8.3  +MOVJ EC00246
SMOVL C00247 BC00247 V=8.3  +MOVJ EC00247
ARCOF
SMOVL C00248 BC00248 V=800.0  +MOVJ EC00248
SMOVL C00249 BC00249 V=1000.0  +MOVJ EC00249
SFTOF3D
'EndPath W4887
MOVJ C00250 BC00250 VJ=100.00  +MOVJ EC00250 VJ=100.00
MOVJ C00251 BC00251 VJ=100.00  +MOVJ EC00251 VJ=100.00
MOVJ C00252 BC00252 VJ=100.00  +MOVJ EC00252 VJ=100.00
'R-L Trip
MOVJ C00253 BC00253 VJ=100.00  +MOVJ EC00253 VJ=100.00
CALL JOB:CLEAN-R1_KM_3P
'WireCut
MOVJ C00254 BC00254 VJ=100.00  +MOVJ EC00254 VJ=100.00
'Path S4234
SFTOF3D
MOVJ C00255 BC00255 VJ=100.00  +MOVJ EC00255 VJ=100.00
MOVL C00256 BC00256 V=800.0  +MOVJ EC00256 VJ=100.00
SMOVL C00257 BC00257 V=166.7  +MOVJ EC00257
SREFP 3 C00258 BC00258  +REFP EC00258
CALL JOB:SEARCH-R1-S13D
SET P034 P006
SFTON3D P034
SMOVL C00259 BC00259 V=166.7  +MOVJ EC00259
SMOVL C00260 BC00260 V=166.7  +MOVJ EC00260
SREFP 3 C00261 BC00261  +REFP EC00261
CALL JOB:SEARCH-R1-S13D
SET P034 P006
SFTON3D P034
SMOVL C00262 BC00262 V=166.7  +MOVJ EC00262
MOVL C00263 BC00263 V=800.0  +MOVJ EC00263 VJ=100.00
MOVL C00264 BC00264 V=1000.0  +MOVJ EC00264 VJ=100.00
'EndPath S4234
'Path S4235
SFTOF3D
MOVJ C00265 BC00265 VJ=100.00  +MOVJ EC00265 VJ=100.00
MOVL C00266 BC00266 V=800.0  +MOVJ EC00266 VJ=100.00
SMOVL C00267 BC00267 V=166.7  +MOVJ EC00267
SREFP 3 C00268 BC00268  +REFP EC00268
CALL JOB:SEARCH-R1-S13D
SET P033 P006
SFTON3D P033
SMOVL C00269 BC00269 V=166.7  +MOVJ EC00269
SMOVL C00270 BC00270 V=166.7  +MOVJ EC00270
SREFP 3 C00271 BC00271  +REFP EC00271
CALL JOB:SEARCH-R1-S13D
SET P033 P006
SFTON3D P033
SMOVL C00272 BC00272 V=166.7  +MOVJ EC00272
MOVL C00273 BC00273 V=800.0  +MOVJ EC00273 VJ=100.00
MOVL C00274 BC00274 V=1000.0  +MOVJ EC00274 VJ=100.00
'EndPath S4235
'Path S4236
SFTOF3D
MOVJ C00275 BC00275 VJ=100.00  +MOVJ EC00275 VJ=100.00
MOVL C00276 BC00276 V=800.0  +MOVJ EC00276 VJ=100.00
SMOVL C00277 BC00277 V=166.7  +MOVJ EC00277
SREFP 3 C00278 BC00278  +REFP EC00278
CALL JOB:SEARCH-R1-S13D
SET P024 P006
SFTON3D P024
SMOVL C00279 BC00279 V=166.7  +MOVJ EC00279
SMOVL C00280 BC00280 V=166.7  +MOVJ EC00280
SREFP 3 C00281 BC00281  +REFP EC00281
CALL JOB:SEARCH-R1-S13D
SET P024 P006
SFTON3D P024
SMOVL C00282 BC00282 V=166.7  +MOVJ EC00282
MOVL C00283 BC00283 V=800.0  +MOVJ EC00283 VJ=100.00
MOVL C00284 BC00284 V=1000.0  +MOVJ EC00284 VJ=100.00
'EndPath S4236
'Path S4237
SFTOF3D
MOVJ C00285 BC00285 VJ=100.00  +MOVJ EC00285 VJ=100.00
MOVL C00286 BC00286 V=800.0  +MOVJ EC00286 VJ=100.00
SMOVL C00287 BC00287 V=166.7  +MOVJ EC00287
SREFP 3 C00288 BC00288  +REFP EC00288
CALL JOB:SEARCH-R1-S13D
SET P023 P006
SFTON3D P023
SMOVL C00289 BC00289 V=166.7  +MOVJ EC00289
SMOVL C00290 BC00290 V=166.7  +MOVJ EC00290
SREFP 3 C00291 BC00291  +REFP EC00291
CALL JOB:SEARCH-R1-S13D
SET P023 P006
SFTON3D P023
SMOVL C00292 BC00292 V=166.7  +MOVJ EC00292
MOVL C00293 BC00293 V=800.0  +MOVJ EC00293 VJ=100.00
MOVL C00294 BC00294 V=1000.0  +MOVJ EC00294 VJ=100.00
'EndPath S4237
'nowe
'Path W4903
SFTOF3D
SFTON3D P024
MOVJ C00295 BC00295 VJ=100.00  +MOVJ EC00295 VJ=100.00
SMOVL C00296 BC00296 V=800.0  +MOVJ EC00296
SMOVL C00297 BC00297 V=150.0 PL=0  +MOVJ EC00297
MACRO1 MJ#(0) ARGF14
ARCON
SMOVL C00298 BC00298 V=9.2  +MOVJ EC00298
SFTON3D P023
SMOVL C00299 BC00299 V=9.2  +MOVJ EC00299
SMOVL C00300 BC00300 V=9.2  +MOVJ EC00300
ARCOF
SMOVL C00301 BC00301 V=800.0  +MOVJ EC00301
SMOVL C00302 BC00302 V=1000.0  +MOVJ EC00302
SFTOF3D
'EndPath W4903
'Path W4906
SFTOF3D
SFTON3D P033
MOVJ C00303 BC00303 VJ=100.00  +MOVJ EC00303 VJ=100.00
SMOVL C00304 BC00304 V=800.0  +MOVJ EC00304
SMOVL C00305 BC00305 V=150.0 PL=0  +MOVJ EC00305
ARCON
SFTON3D P034
SMOVL C00306 BC00306 V=10.7  +MOVJ EC00306
ARCOF
SMOVL C00307 BC00307 V=800.0  +MOVJ EC00307
SMOVL C00308 BC00308 V=1000.0  +MOVJ EC00308
SFTOF3D
'EndPath W4906
MOVJ C00309 BC00309 VJ=100.00  +MOVJ EC00309 VJ=100.00
'WireCut
MOVJ C00310 BC00310 VJ=100.00  +MOVJ EC00310 VJ=100.00
MOVJ C00311 BC00311 VJ=100.00  +MOVJ EC00311 VJ=100.00
MOVJ C00312 BC00312 VJ=100.00  +MOVJ EC00312 VJ=100.00
MOVJ C00313 BC00313 VJ=100.00  +MOVJ EC00313 VJ=100.00
CALL JOB:CLEAN-R1_KM_3P
MOVJ C00314 BC00314 VJ=100.00  +MOVJ EC00314 VJ=100.00
MOVJ C00315 BC00315 VJ=100.00  +MOVJ EC00315 VJ=100.00
'L-R Trip
'Path S4249
SFTOF3D
MOVJ C00316 BC00316 VJ=100.00  +MOVJ EC00316 VJ=100.00
MOVL C00317 BC00317 V=800.0  +MOVJ EC00317 VJ=100.00
SMOVL C00318 BC00318 V=166.7  +MOVJ EC00318
SREFP 3 C00319 BC00319  +REFP EC00319
CALL JOB:SEARCH-R1-S13D
SET P036 P006
SFTON3D P036
SMOVL C00320 BC00320 V=166.7  +MOVJ EC00320
SMOVL C00321 BC00321 V=166.7  +MOVJ EC00321
SREFP 3 C00322 BC00322  +REFP EC00322
CALL JOB:SEARCH-R1-S13D
SET P036 P006
SFTON3D P036
SMOVL C00323 BC00323 V=166.7  +MOVJ EC00323
MOVL C00324 BC00324 V=800.0  +MOVJ EC00324 VJ=100.00
MOVL C00325 BC00325 V=1000.0  +MOVJ EC00325 VJ=100.00
'EndPath S4249
'Path S4250
SFTOF3D
MOVJ C00326 BC00326 VJ=100.00  +MOVJ EC00326 VJ=100.00
MOVL C00327 BC00327 V=800.0  +MOVJ EC00327 VJ=100.00
SMOVL C00328 BC00328 V=166.7  +MOVJ EC00328
SREFP 3 C00329 BC00329  +REFP EC00329
CALL JOB:SEARCH-R1-S13D
SET P035 P006
SFTON3D P035
SMOVL C00330 BC00330 V=166.7  +MOVJ EC00330
SMOVL C00331 BC00331 V=166.7  +MOVJ EC00331
SREFP 3 C00332 BC00332  +REFP EC00332
CALL JOB:SEARCH-R1-S13D
SET P035 P006
SFTON3D P035
SMOVL C00333 BC00333 V=166.7  +MOVJ EC00333
MOVL C00334 BC00334 V=800.0  +MOVJ EC00334 VJ=100.00
MOVL C00335 BC00335 V=1000.0  +MOVJ EC00335 VJ=100.00
'EndPath S4250
'Path S4251
SFTOF3D
MOVJ C00336 BC00336 VJ=100.00  +MOVJ EC00336 VJ=100.00
MOVL C00337 BC00337 V=800.0  +MOVJ EC00337 VJ=100.00
SMOVL C00338 BC00338 V=166.7  +MOVJ EC00338
SREFP 3 C00339 BC00339  +REFP EC00339
CALL JOB:SEARCH-R1-S13D
SET P026 P006
SFTON3D P026
SMOVL C00340 BC00340 V=166.7  +MOVJ EC00340
SMOVL C00341 BC00341 V=166.7  +MOVJ EC00341
SREFP 3 C00342 BC00342  +REFP EC00342
CALL JOB:SEARCH-R1-S13D
SET P026 P006
SFTON3D P026
SMOVL C00343 BC00343 V=166.7  +MOVJ EC00343
MOVL C00344 BC00344 V=800.0  +MOVJ EC00344 VJ=100.00
MOVL C00345 BC00345 V=1000.0  +MOVJ EC00345 VJ=100.00
'EndPath S4251
'Path S4252
SFTOF3D
MOVJ C00346 BC00346 VJ=100.00  +MOVJ EC00346 VJ=100.00
MOVL C00347 BC00347 V=800.0  +MOVJ EC00347 VJ=100.00
SMOVL C00348 BC00348 V=166.7  +MOVJ EC00348
SREFP 3 C00349 BC00349  +REFP EC00349
CALL JOB:SEARCH-R1-S13D
SET P025 P006
SFTON3D P025
SMOVL C00350 BC00350 V=166.7  +MOVJ EC00350
SMOVL C00351 BC00351 V=166.7  +MOVJ EC00351
SREFP 3 C00352 BC00352  +REFP EC00352
CALL JOB:SEARCH-R1-S13D
SET P025 P006
SFTON3D P025
SMOVL C00353 BC00353 V=166.7  +MOVJ EC00353
MOVL C00354 BC00354 V=800.0  +MOVJ EC00354 VJ=100.00
MOVL C00355 BC00355 V=1000.0  +MOVJ EC00355 VJ=100.00
'EndPath S4252
'Path W4907
SFTOF3D
SFTON3D P026
MOVJ C00356 BC00356 VJ=100.00  +MOVJ EC00356 VJ=100.00
SMOVL C00357 BC00357 V=800.0  +MOVJ EC00357
SMOVL C00358 BC00358 V=150.0 PL=0  +MOVJ EC00358
ARCON
SFTON3D P025
SMOVL C00359 BC00359 V=11.7  +MOVJ EC00359
ARCOF
SMOVL C00360 BC00360 V=800.0  +MOVJ EC00360
SMOVL C00361 BC00361 V=1000.0  +MOVJ EC00361
SFTOF3D
'EndPath W4907
'Path W4908
SFTOF3D
SFTON3D P035
MOVJ C00362 BC00362 VJ=100.00  +MOVJ EC00362 VJ=100.00
SMOVL C00363 BC00363 V=800.0  +MOVJ EC00363
SMOVL C00364 BC00364 V=150.0 PL=0  +MOVJ EC00364
ARCON
SFTON3D P036
SMOVL C00365 BC00365 V=11.7  +MOVJ EC00365
ARCOF
SMOVL C00366 BC00366 V=800.0  +MOVJ EC00366
SMOVL C00367 BC00367 V=1000.0  +MOVJ EC00367
SFTOF3D
'EndPath W4908
MOVJ C00368 BC00368 VJ=100.00  +MOVJ EC00368 VJ=100.00
MOVJ C00369 BC00369 VJ=100.00  +MOVJ EC00369 VJ=100.00
CALL JOB:CLEAN-R1_KM_3P
MOVJ C00370 BC00370 VJ=100.00  +MOVJ EC00370 VJ=100.00
MOVJ C00371 BC00371 VJ=100.00  +MOVJ EC00371 VJ=100.00
MOVJ C00372 BC00372 VJ=100.00  +MOVJ EC00372 VJ=100.00
'Path S4888
SFTOF3D
MOVJ C00373 BC00373 VJ=100.00  +MOVJ EC00373 VJ=100.00
MOVL C00374 BC00374 V=800.0  +MOVJ EC00374 VJ=100.00
SMOVL C00375 BC00375 V=166.7  +MOVJ EC00375
SREFP 3 C00376 BC00376  +REFP EC00376
CALL JOB:SEARCH-R1-S13D
SET P044 P006
SFTON3D P044
SMOVL C00377 BC00377 V=166.7  +MOVJ EC00377
SMOVL C00378 BC00378 V=166.7  +MOVJ EC00378
SREFP 3 C00379 BC00379  +REFP EC00379
CALL JOB:SEARCH-R1-S13D
SET P044 P006
SFTON3D P044
SMOVL C00380 BC00380 V=166.7  +MOVJ EC00380
MOVL C00381 BC00381 V=800.0  +MOVJ EC00381 VJ=100.00
MOVL C00382 BC00382 V=1000.0  +MOVJ EC00382 VJ=100.00
'EndPath S4888
'Path S4889
SFTOF3D
MOVJ C00383 BC00383 VJ=100.00  +MOVJ EC00383 VJ=100.00
MOVL C00384 BC00384 V=800.0  +MOVJ EC00384 VJ=100.00
SMOVL C00385 BC00385 V=166.7  +MOVJ EC00385
SREFP 3 C00386 BC00386  +REFP EC00386
CALL JOB:SEARCH-R1-S13D
SET P043 P006
SFTON3D P043
SMOVL C00387 BC00387 V=166.7  +MOVJ EC00387
SMOVL C00388 BC00388 V=166.7  +MOVJ EC00388
SREFP 3 C00389 BC00389  +REFP EC00389
CALL JOB:SEARCH-R1-S13D
SET P043 P006
SFTON3D P043
SMOVL C00390 BC00390 V=166.7  +MOVJ EC00390
MOVL C00391 BC00391 V=800.0  +MOVJ EC00391 VJ=100.00
MOVL C00392 BC00392 V=1000.0  +MOVJ EC00392 VJ=100.00
'EndPath S4889
MOVJ C00393 BC00393 VJ=100.00  +MOVJ EC00393 VJ=100.00
MOVJ C00394 BC00394 VJ=100.00  +MOVJ EC00394 VJ=100.00
MOVJ C00395 BC00395 VJ=100.00  +MOVJ EC00395 VJ=100.00
MOVJ C00396 BC00396 VJ=100.00  +MOVJ EC00396 VJ=100.00
'Path S4899
SFTOF3D
MOVJ C00397 BC00397 VJ=100.00  +MOVJ EC00397 VJ=100.00
MOVL C00398 BC00398 V=800.0  +MOVJ EC00398 VJ=100.00
SMOVL C00399 BC00399 V=166.7  +MOVJ EC00399
SREFP 3 C00400 BC00400  +REFP EC00400
CALL JOB:SEARCH-R1-S13D
SET P046 P006
SFTON3D P046
SMOVL C00401 BC00401 V=166.7  +MOVJ EC00401
SMOVL C00402 BC00402 V=166.7  +MOVJ EC00402
SREFP 3 C00403 BC00403  +REFP EC00403
CALL JOB:SEARCH-R1-S13D
SET P046 P006
SFTON3D P046
SMOVL C00404 BC00404 V=166.7  +MOVJ EC00404
MOVL C00405 BC00405 V=800.0  +MOVJ EC00405 VJ=100.00
MOVL C00406 BC00406 V=1000.0  +MOVJ EC00406 VJ=100.00
'EndPath S4899
MOVJ C00407 BC00407 VJ=100.00  +MOVJ EC00407 VJ=100.00
'Path S4888
SFTOF3D
MOVJ C00408 BC00408 VJ=100.00  +MOVJ EC00408 VJ=100.00
MOVL C00409 BC00409 V=800.0  +MOVJ EC00409 VJ=100.00
SMOVL C00410 BC00410 V=166.7  +MOVJ EC00410
SREFP 3 C00411 BC00411  +REFP EC00411
CALL JOB:SEARCH-R1-S13D
SET P028 P006
SFTON3D P028
SMOVL C00412 BC00412 V=166.7  +MOVJ EC00412
SMOVL C00413 BC00413 V=166.7  +MOVJ EC00413
SREFP 3 C00414 BC00414  +REFP EC00414
CALL JOB:SEARCH-R1-S13D
SET P028 P006
SFTON3D P028
SMOVL C00415 BC00415 V=166.7  +MOVJ EC00415
MOVL C00416 BC00416 V=800.0  +MOVJ EC00416 VJ=100.00
MOVL C00417 BC00417 V=1000.0  +MOVJ EC00417 VJ=100.00
'EndPath S4888
'Path S4889
SFTOF3D
MOVJ C00418 BC00418 VJ=100.00  +MOVJ EC00418 VJ=100.00
MOVL C00419 BC00419 V=800.0  +MOVJ EC00419 VJ=100.00
SMOVL C00420 BC00420 V=166.7  +MOVJ EC00420
SREFP 3 C00421 BC00421  +REFP EC00421
CALL JOB:SEARCH-R1-S13D
SET P027 P006
SFTON3D P027
SMOVL C00422 BC00422 V=166.7  +MOVJ EC00422
SMOVL C00423 BC00423 V=166.7  +MOVJ EC00423
SREFP 3 C00424 BC00424  +REFP EC00424
CALL JOB:SEARCH-R1-S13D
SET P027 P006
SFTON3D P027
SMOVL C00425 BC00425 V=166.7  +MOVJ EC00425
MOVL C00426 BC00426 V=800.0  +MOVJ EC00426 VJ=100.00
MOVL C00427 BC00427 V=1000.0  +MOVJ EC00427 VJ=100.00
'EndPath S4889
'Path W4890
SFTOF3D
SFTON3D P027
MOVJ C00428 BC00428 VJ=100.00  +MOVJ EC00428 VJ=100.00
SMOVL C00429 BC00429 V=800.0  +MOVJ EC00429
SMOVL C00430 BC00430 V=150.0 PL=0  +MOVJ EC00430
MACRO1 MJ#(0) ARGF6
ARCON
SMOVL C00431 BC00431 V=6.7  +MOVJ EC00431
SFTON3D P028
SMOVL C00432 BC00432 V=10.0  +MOVJ EC00432
ARCOF
SMOVL C00433 BC00433 V=800.0  +MOVJ EC00433
SMOVL C00434 BC00434 V=1000.0  +MOVJ EC00434
SFTOF3D
'EndPath W4890
MOVJ C00435 BC00435 VJ=100.00  +MOVJ EC00435 VJ=100.00
MOVJ C00436 BC00436 VJ=100.00  +MOVJ EC00436 VJ=100.00
MOVJ C00437 BC00437 VJ=100.00  +MOVJ EC00437 VJ=100.00
MOVJ C00438 BC00438 VJ=100.00  +MOVJ EC00438 VJ=100.00
MOVJ C00439 BC00439 VJ=100.00  +MOVJ EC00439 VJ=100.00
'Path W4900
SFTOF3D
SFTON3D P043
MOVJ C00440 BC00440 VJ=100.00  +MOVJ EC00440 VJ=100.00
SMOVL C00441 BC00441 V=800.0  +MOVJ EC00441
SMOVL C00442 BC00442 V=150.0 PL=0  +MOVJ EC00442
MACRO1 MJ#(0) ARGF14
ARCON
SFTON3D P044
SMOVL C00443 BC00443 V=10.0  +MOVJ EC00443
SMOVL C00444 BC00444 V=10.0  +MOVJ EC00444
ARCOF
SMOVL C00445 BC00445 V=800.0  +MOVJ EC00445
SMOVL C00446 BC00446 V=1000.0  +MOVJ EC00446
SFTOF3D
'EndPath W4900
MOVJ C00447 BC00447 VJ=100.00  +MOVJ EC00447 VJ=100.00
MOVJ C00448 BC00448 VJ=100.00  +MOVJ EC00448 VJ=100.00
MOVJ C00449 BC00449 VJ=100.00  +MOVJ EC00449 VJ=100.00
MOVJ C00450 BC00450 VJ=100.00  +MOVJ EC00450 VJ=100.00
MOVJ C00451 BC00451 VJ=100.00  +MOVJ EC00451 VJ=100.00
'Path W4898
SFTOF3D
SFTON3D P046
MOVJ C00452 BC00452 VJ=100.00  +MOVJ EC00452 VJ=100.00
SMOVL C00453 BC00453 V=800.0  +MOVJ EC00453
SMOVL C00454 BC00454 V=150.0 PL=0  +MOVJ EC00454
ARCON
SMOVL C00455 BC00455 V=10.0  +MOVJ EC00455
SMOVL C00456 BC00456 V=10.0  +MOVJ EC00456
ARCOF
SMOVL C00457 BC00457 V=800.0  +MOVJ EC00457
SMOVL C00458 BC00458 V=1000.0  +MOVJ EC00458
SFTOF3D
'EndPath W4898
MOVJ C00459 BC00459 VJ=100.00  +MOVJ EC00459 VJ=100.00
MOVJ C00460 BC00460 VJ=100.00  +MOVJ EC00460 VJ=100.00
MOVJ C00461 BC00461 VJ=100.00  +MOVJ EC00461 VJ=100.00
MOVJ C00462 BC00462 VJ=100.00  +MOVJ EC00462 VJ=100.00
MOVJ C00463 BC00463 VJ=100.00  +MOVJ EC00463 VJ=100.00
END
